	//Sorties
	"DB_BIBLIOTHEQUE".Mobile[#index].Pos[1].Sort1[0] := "I_CP_BD2EVS10_T63";
	"DB_BIBLIOTHEQUE".Mobile[#index].Pos[1].Sort0[0] := "I_CP_BD2EVS10_TVS20";
	"DB_BIBLIOTHEQUE".Mobile[#index].Pos[1].Sort0_Pr_Fin_Pos[0] := "I_CP_BD2EVS10_T63";
	"DB_BIBLIOTHEQUE".Mobile[#index].Pos[1].Sort0_Pr_Fin_Pos[1] := "I_CP_BD2EVS10_TVS20";


	#index := #index + 1;
	(*
	           ╔═══════════╗
	           ║    TR11   ║
	           ╚═══════════╝
	*)
	//++++++++++++++++++++++87++++++++++++++++++++++++++++++\\
	"DB_BIBLIOTHEQUE".Mobile[#index].Noeud := TRUE;

	"DB_BIBLIOTHEQUE".Mobile[#index].Nom := 'TR11';
	"DB_BIBLIOTHEQUE".Mobile[#index].Mob_Suiv[0] := "Index_Mobile"('TR1TR11');
	"DB_BIBLIOTHEQUE".Mobile[#index].Mob_Suiv[1] := "Index_Mobile"('TR2TR11');
	"DB_BIBLIOTHEQUE".Mobile[#index].Mob_Prec[0] := "Index_Mobile"('BD1ER10');
	"DB_BIBLIOTHEQUE".Mobile[#index].Mob_Prec[1] := "Index_Mobile"('BD1EVS10');

	"DB_BIBLIOTHEQUE".Mobile[#index].Pos[0].Nom := '_VERS_TR1TR2TR11';
	"DB_BIBLIOTHEQUE".Mobile[#index].Pos[0].Mob_Suiv[0] := "Index_Mobile"('TR1TR11');
	"DB_BIBLIOTHEQUE".Mobile[#index].Pos[0].Mob_Suiv[1] := "Index_Mobile"('TR2TR11');


	//"DB_BIBLIOTHEQUE".Mobile[#index].Pass_Mat := "RPM_TR11";


	// Entrées avant pos
	"DB_BIBLIOTHEQUE".Mobile[#index].Pos[0].Entr0_Av_Pos[0] := "I_RD_DISJ_TR11";

	// Entrées apres pos
	"DB_BIBLIOTHEQUE".Mobile[#index].Pos[0].Entr0_Ap_Pos[0] := "I_RB_TR11";
	"DB_BIBLIOTHEQUE".Mobile[#index].Pos[0].Entr0_Ap_Pos[1] := "I_RD_DISJ_TR11";


	//"DB_BIBLIOTHEQUE".Mobile[#index].Pos[0].Entr1_Ap_Pos[0] := "I_RR_TR11";
	"DB_BIBLIOTHEQUE".Mobile[#index].Pos[0].Entr1_Ap_Pos[0] := "I_RM_TR11";

	// Entrées fin pos
	//"DB_BIBLIOTHEQUE".Mobile[#index].Pos[0].Entr0_Ap_Fin_Pos[0]:="I_RM_TR11";

	// Sorties
	"DB_BIBLIOTHEQUE".Mobile[#index].Pos[0].Sort1[0] := "I_CM_TR11";
	"DB_BIBLIOTHEQUE".Mobile[#index].Pos[0].Sort0_Pr_Fin_Pos[0] := "I_CM_TR11";


	#index := #index + 1;
	(*
	           ╔═══════════╗
	           ║   TR1TR11 ║
	           ╚═══════════╝
	*)
	//++++++++++++++++++++++88++++++++++++++++++++++++++++++\\



	"DB_BIBLIOTHEQUE".Mobile[#index].Nom := 'TR1TR11';
	"DB_BIBLIOTHEQUE".Mobile[#index].Mob_Suiv[0] := "Index_Mobile"('BD1TR11');
	"DB_BIBLIOTHEQUE".Mobile[#index].Mob_Prec[0] := "Index_Mobile"('TR11');

	"DB_BIBLIOTHEQUE".Mobile[#index].Pos[0].Nom := '_CLOSE';
	//"DB_BIBLIOTHEQUE".Mobile[#index].Pos[0].Mob_Suiv[0] := "Index_Mobile"('BD1TR11');
	"DB_BIBLIOTHEQUE".Mobile[#index].Pos[1].Nom := '_OPEN';
	"DB_BIBLIOTHEQUE".Mobile[#index].Pos[1].Mob_Suiv[0] := "Index_Mobile"('BD1TR11');


	//position fermeture
	"DB_BIBLIOTHEQUE".Mobile[#index].Pos[0].Entr0_Ap_Pos[0] := "I_RPO_TR1TR11";
	"DB_BIBLIOTHEQUE".Mobile[#index].Pos[0].Entr1_Ap_Pos[0] := "I_RPF_TR1TR11";
	"DB_BIBLIOTHEQUE".Mobile[#index].Pos[0].Sort0[0] := "I_CO_TR1TR11";
	"DB_BIBLIOTHEQUE".Mobile[#index].Pos[0].Sort0_Pr_Fin_Pos[0] := "I_CO_TR1TR11";

	//position ouverture
	"DB_BIBLIOTHEQUE".Mobile[#index].Pos[1].Entr0_Ap_Pos[0] := "I_RPF_TR1TR11";
	"DB_BIBLIOTHEQUE".Mobile[#index].Pos[1].Entr1_Ap_Pos[0] := "I_RPO_TR1TR11";
	"DB_BIBLIOTHEQUE".Mobile[#index].Pos[1].Sort1[0] := "I_CO_TR1TR11";
	"DB_BIBLIOTHEQUE".Mobile[#index].Pos[1].Sort0_Pr_Fin_Pos[0] := "I_CO_TR1TR11";



	#index := #index + 1;
	(*
	           ╔═══════════╗
	           ║   TR2TR11 ║
	           ╚═══════════╝
	*)
	//++++++++++++++++++++++89++++++++++++++++++++++++++++++\\


	"DB_BIBLIOTHEQUE".Mobile[#index].Nom := 'TR2TR11';
	"DB_BIBLIOTHEQUE".Mobile[#index].Mob_Suiv[0] := "Index_Mobile"('BD2TR11');
	"DB_BIBLIOTHEQUE".Mobile[#index].Mob_Prec[0] := "Index_Mobile"('TR11');

	"DB_BIBLIOTHEQUE".Mobile[#index].Pos[0].Nom := '_CLOSE';
	//"DB_BIBLIOTHEQUE".Mobile[#index].Pos[0].Mob_Suiv[0] := "Index_Mobile"('BD2TR11');
	"DB_BIBLIOTHEQUE".Mobile[#index].Pos[1].Nom := '_OPEN';
	"DB_BIBLIOTHEQUE".Mobile[#index].Pos[1].Mob_Suiv[0] := "Index_Mobile"('BD2TR11');


	//position fermeture
	"DB_BIBLIOTHEQUE".Mobile[#index].Pos[0].Entr0_Ap_Pos[0] := "I_RPO_TR2TR11";
	"DB_BIBLIOTHEQUE".Mobile[#index].Pos[0].Entr1_Ap_Pos[0] := "I_RPF_TR2TR11";
	"DB_BIBLIOTHEQUE".Mobile[#index].Pos[0].Sort0[0] := "I_CO_TR2TR11";
	"DB_BIBLIOTHEQUE".Mobile[#index].Pos[0].Sort0_Pr_Fin_Pos[0] := "I_CO_TR2TR11";

	//position ouverture
	"DB_BIBLIOTHEQUE".Mobile[#index].Pos[1].Entr0_Ap_Pos[0] := "I_RPF_TR2TR11";
	"DB_BIBLIOTHEQUE".Mobile[#index].Pos[1].Entr1_Ap_Pos[0] := "I_RPO_TR2TR11";
	"DB_BIBLIOTHEQUE".Mobile[#index].Pos[1].Sort1[0] := "I_CO_TR2TR11";
	"DB_BIBLIOTHEQUE".Mobile[#index].Pos[1].Sort0_Pr_Fin_Pos[0] := "I_CO_TR2TR11";



	#index := #index + 1;
	(*
	           ╔═══════════╗
	           ║  BD1TR11  ║
	           ╚═══════════╝
	*)
	//++++++++++++++++++++++90++++++++++++++++++++++++++++++\\
	"DB_BIBLIOTHEQUE".Mobile[#index].Noeud := TRUE;


	"DB_BIBLIOTHEQUE".Mobile[#index].Nom := 'BD1TR11';
	"DB_BIBLIOTHEQUE".Mobile[#index].Mob_Suiv[0] := "Index_Mobile"('S21');
	"DB_BIBLIOTHEQUE".Mobile[#index].Mob_Suiv[1] := "Index_Mobile"('TR12');
	"DB_BIBLIOTHEQUE".Mobile[#index].Mob_Prec[0] := "Index_Mobile"('TR1TR11');


	"DB_BIBLIOTHEQUE".Mobile[#index].Pos[0].Nom := '_VERS_S21';
	"DB_BIBLIOTHEQUE".Mobile[#index].Pos[0].Mob_Suiv[0] := "Index_Mobile"('S21');
	"DB_BIBLIOTHEQUE".Mobile[#index].Pos[1].Nom := '_VERS_TR12';
	"DB_BIBLIOTHEQUE".Mobile[#index].Pos[1].Mob_Suiv[0] := "Index_Mobile"('TR12');




	//Entrées
	"DB_BIBLIOTHEQUE".Mobile[#index].Pos[0].Entr0_Ap_Pos[0] := "I_RP_BD1TR11_TR12";
	"DB_BIBLIOTHEQUE".Mobile[#index].Pos[0].Entr1_Ap_Pos[0] := "I_RP_BD1TR11_S21";
	"DB_BIBLIOTHEQUE".Mobile[#index].Pos[0].Sort1[0] := "I_CP_BD1TR11_S21";
	"DB_BIBLIOTHEQUE".Mobile[#index].Pos[0].Sort0[0] := "I_CP_BD1TR11_TR12";
	"DB_BIBLIOTHEQUE".Mobile[#index].Pos[0].Sort0_Pr_Fin_Pos[0] := "I_CP_BD1TR11_TR12";
	"DB_BIBLIOTHEQUE".Mobile[#index].Pos[0].Sort0_Pr_Fin_Pos[1] := "I_CP_BD1TR11_S21";

	"DB_BIBLIOTHEQUE".Mobile[#index].Pos[1].Entr0_Ap_Pos[1] := "I_RP_BD1TR11_S21";
	"DB_BIBLIOTHEQUE".Mobile[#index].Pos[1].Entr1_Ap_Pos[1] := "I_RP_BD1TR11_TR12";

	//Sorties
	"DB_BIBLIOTHEQUE".Mobile[#index].Pos[1].Sort1[0] := "I_CP_BD1TR11_TR12";
	"DB_BIBLIOTHEQUE".Mobile[#index].Pos[1].Sort0[0] := "I_CP_BD1TR11_S21";
	"DB_BIBLIOTHEQUE".Mobile[#index].Pos[1].Sort0_Pr_Fin_Pos[0] := "I_CP_BD1TR11_TR12";
	"DB_BIBLIOTHEQUE".Mobile[#index].Pos[1].Sort0_Pr_Fin_Pos[1] := "I_CP_BD1TR11_S21";


	#index := #index + 1;
	(*
	           ╔═══════════╗
	           ║  BD2TR11  ║
	           ╚═══════════╝
	*)
	//++++++++++++++++++++++91++++++++++++++++++++++++++++++\\
	"DB_BIBLIOTHEQUE".Mobile[#index].Noeud := TRUE;


	"DB_BIBLIOTHEQUE".Mobile[#index].Nom := 'BD2TR11';
	"DB_BIBLIOTHEQUE".Mobile[#index].Mob_Suiv[0] := "Index_Mobile"('S23');
	"DB_BIBLIOTHEQUE".Mobile[#index].Mob_Suiv[1] := "Index_Mobile"('TR13');
	"DB_BIBLIOTHEQUE".Mobile[#index].Mob_Prec[0] := "Index_Mobile"('TR2TR11');


	"DB_BIBLIOTHEQUE".Mobile[#index].Pos[0].Nom := '_VERS_S23';
	"DB_BIBLIOTHEQUE".Mobile[#index].Pos[0].Mob_Suiv[0] := "Index_Mobile"('S23');
	"DB_BIBLIOTHEQUE".Mobile[#index].Pos[1].Nom := '_VERS_TR13';
	"DB_BIBLIOTHEQUE".Mobile[#index].Pos[1].Mob_Suiv[0] := "Index_Mobile"('TR13');




	//Entrées
	"DB_BIBLIOTHEQUE".Mobile[#index].Pos[0].Entr0_Ap_Pos[0] := "I_RP_BD2TR11_TR13";
	"DB_BIBLIOTHEQUE".Mobile[#index].Pos[0].Entr1_Ap_Pos[0] := "I_RP_BD2TR11_S23";
	"DB_BIBLIOTHEQUE".Mobile[#index].Pos[0].Sort1[0] := "I_CP_BD2TR11_S23";
	"DB_BIBLIOTHEQUE".Mobile[#index].Pos[0].Sort0[0] := "I_CP_BD2TR11_TR13";
	"DB_BIBLIOTHEQUE".Mobile[#index].Pos[0].Sort0_Pr_Fin_Pos[0] := "I_CP_BD2TR11_TR13";
	"DB_BIBLIOTHEQUE".Mobile[#index].Pos[0].Sort0_Pr_Fin_Pos[1] := "I_CP_BD2TR11_S23";

	"DB_BIBLIOTHEQUE".Mobile[#index].Pos[1].Entr0_Ap_Pos[1] := "I_RP_BD2TR11_S23";
	"DB_BIBLIOTHEQUE".Mobile[#index].Pos[1].Entr1_Ap_Pos[1] := "I_RP_BD2TR11_TR13";

	//Sorties
	"DB_BIBLIOTHEQUE".Mobile[#index].Pos[1].Sort1[0] := "I_CP_BD2TR11_TR13";
	"DB_BIBLIOTHEQUE".Mobile[#index].Pos[1].Sort0[0] := "I_CP_BD2TR11_S23";
	"DB_BIBLIOTHEQUE".Mobile[#index].Pos[1].Sort0_Pr_Fin_Pos[0] := "I_CP_BD2TR11_TR13";
	"DB_BIBLIOTHEQUE".Mobile[#index].Pos[1].Sort0_Pr_Fin_Pos[1] := "I_CP_BD2TR11_S23";


	#index := #index + 1;
	(*
	           ╔═══════════╗
	           ║    TR12   ║
	           ╚═══════════╝
	*)
	//++++++++++++++++++++++92++++++++++++++++++++++++++++++\\


	"DB_BIBLIOTHEQUE".Mobile[#index].Nom := 'TR12';
	"DB_BIBLIOTHEQUE".Mobile[#index].Mob_Suiv[0] := "Index_Mobile"('S22');
	"DB_BIBLIOTHEQUE".Mobile[#index].Mob_Prec[0] := "Index_Mobile"('BD1TR11');

	"DB_BIBLIOTHEQUE".Mobile[#index].Pos[0].Nom := '_VERSS22';
	"DB_BIBLIOTHEQUE".Mobile[#index].Pos[0].Mob_Suiv[0] := "Index_Mobile"('S22');


	//"DB_BIBLIOTHEQUE".Mobile[#index].Pass_Mat := "RPM_TR12";


	// Entrées avant pos
	"DB_BIBLIOTHEQUE".Mobile[#index].Pos[0].Entr0_Av_Pos[0] := "I_RD_DISJ_TR12";

	// Entrées apres pos
	"DB_BIBLIOTHEQUE".Mobile[#index].Pos[0].Entr0_Ap_Pos[0] := "I_RB_TR12";
	"DB_BIBLIOTHEQUE".Mobile[#index].Pos[0].Entr0_Ap_Pos[1] := "I_RD_DISJ_TR12";


	//"DB_BIBLIOTHEQUE".Mobile[#index].Pos[0].Entr1_Ap_Pos[0] := "I_RR_TR12";
	"DB_BIBLIOTHEQUE".Mobile[#index].Pos[0].Entr1_Ap_Pos[0] := "I_RM_TR12";

	// Entrées fin pos
	//"DB_BIBLIOTHEQUE".Mobile[#index].Pos[0].Entr0_Ap_Fin_Pos[0]:="I_RM_TR12";

	// Sorties
	"DB_BIBLIOTHEQUE".Mobile[#index].Pos[0].Sort1[0] := "I_CM_TR12";
	"DB_BIBLIOTHEQUE".Mobile[#index].Pos[0].Sort0_Pr_Fin_Pos[0] := "I_CM_TR12";


	#index := #index + 1;
	(*
	           ╔═══════════╗
	           ║    TR13   ║
	           ╚═══════════╝
	*)
	//++++++++++++++++++++++93++++++++++++++++++++++++++++++\\


	"DB_BIBLIOTHEQUE".Mobile[#index].Nom := 'TR13';
	"DB_BIBLIOTHEQUE".Mobile[#index].Mob_Suiv[0] := "Index_Mobile"('S24');
	"DB_BIBLIOTHEQUE".Mobile[#index].Mob_Prec[0] := "Index_Mobile"('BD2TR11');

	"DB_BIBLIOTHEQUE".Mobile[#index].Pos[0].Nom := '_VERSS24';
	"DB_BIBLIOTHEQUE".Mobile[#index].Pos[0].Mob_Suiv[0] := "Index_Mobile"('S24');

	//"DB_BIBLIOTHEQUE".Mobile[#index].Pass_Mat := "RPM_TR13";


	// Entrées avant pos
	"DB_BIBLIOTHEQUE".Mobile[#index].Pos[0].Entr0_Av_Pos[0] := "I_RD_DISJ_TR13";

	// Entrées apres pos
	"DB_BIBLIOTHEQUE".Mobile[#index].Pos[0].Entr0_Ap_Pos[0] := "I_RB_TR13";
	"DB_BIBLIOTHEQUE".Mobile[#index].Pos[0].Entr0_Ap_Pos[1] := "I_RD_DISJ_TR13";


	//"DB_BIBLIOTHEQUE".Mobile[#index].Pos[0].Entr1_Ap_Pos[0] := "I_RR_TR13";
	"DB_BIBLIOTHEQUE".Mobile[#index].Pos[0].Entr1_Ap_Pos[0] := "I_RM_TR13";

	// Entrées fin pos
	//"DB_BIBLIOTHEQUE".Mobile[#index].Pos[0].Entr0_Ap_Fin_Pos[0]:="I_RM_TR13";

	// Sorties
	"DB_BIBLIOTHEQUE".Mobile[#index].Pos[0].Sort1[0] := "I_CM_TR13";
	"DB_BIBLIOTHEQUE".Mobile[#index].Pos[0].Sort0_Pr_Fin_Pos[0] := "I_CM_TR13";


	#index := #index + 1;
	(*
	           ╔═══════════╗
	           ║   VAS21   ║
	           ╚═══════════╝
	*)
	//++++++++++++++++++++++94++++++++++++++++++++++++++++++\\



	"DB_BIBLIOTHEQUE".Mobile[#index].Nom := 'VAS21';
	"DB_BIBLIOTHEQUE".Mobile[#index].Mob_Suiv[0] := "Index_Mobile"('TVS212');
	"DB_BIBLIOTHEQUE".Mobile[#index].Mob_Prec[0] := "Index_Mobile"('S21');

	"DB_BIBLIOTHEQUE".Mobile[#index].Pos[0].Nom := '_CLOSE';
	//"DB_BIBLIOTHEQUE".Mobile[#index].Pos[0].Mob_Suiv[0] := "Index_Mobile"('TVS212');
	"DB_BIBLIOTHEQUE".Mobile[#index].Pos[1].Nom := '_OPEN';
	"DB_BIBLIOTHEQUE".Mobile[#index].Pos[1].Mob_Suiv[0] := "Index_Mobile"('TVS212');


	//position fermeture
	"DB_BIBLIOTHEQUE".Mobile[#index].Pos[0].Entr0_Ap_Pos[0] := "I_RPO_VAS21";
	"DB_BIBLIOTHEQUE".Mobile[#index].Pos[0].Entr1_Ap_Pos[0] := "I_RPF_VAS21";
	"DB_BIBLIOTHEQUE".Mobile[#index].Pos[0].Sort0[0] := "I_CO_VAS21";
	"DB_BIBLIOTHEQUE".Mobile[#index].Pos[0].Sort0_Pr_Fin_Pos[0] := "I_CO_VAS21";

	//position ouverture
	"DB_BIBLIOTHEQUE".Mobile[#index].Pos[1].Entr0_Ap_Pos[0] := "I_RPF_VAS21";
	"DB_BIBLIOTHEQUE".Mobile[#index].Pos[1].Entr1_Ap_Pos[0] := "I_RPO_VAS21";
	"DB_BIBLIOTHEQUE".Mobile[#index].Pos[1].Sort1[0] := "I_CO_VAS21";
	"DB_BIBLIOTHEQUE".Mobile[#index].Pos[1].Sort0_Pr_Fin_Pos[0] := "I_CO_VAS21";



	#index := #index + 1;

	(*
	           ╔═══════════╗
	           ║   VAS22   ║
	           ╚═══════════╝
	*)
	//++++++++++++++++++++++95++++++++++++++++++++++++++++++\\



	"DB_BIBLIOTHEQUE".Mobile[#index].Nom := 'VAS22';
	"DB_BIBLIOTHEQUE".Mobile[#index].Mob_Suiv[0] := "Index_Mobile"('TVS22');
	"DB_BIBLIOTHEQUE".Mobile[#index].Mob_Prec[0] := "Index_Mobile"('S22');

	"DB_BIBLIOTHEQUE".Mobile[#index].Pos[0].Nom := '_CLOSE';
	//"DB_BIBLIOTHEQUE".Mobile[#index].Pos[0].Mob_Suiv[0] := "Index_Mobile"('TVS22');
	"DB_BIBLIOTHEQUE".Mobile[#index].Pos[1].Nom := '_OPEN';
	"DB_BIBLIOTHEQUE".Mobile[#index].Pos[1].Mob_Suiv[0] := "Index_Mobile"('TVS22');


	//position fermeture
	"DB_BIBLIOTHEQUE".Mobile[#index].Pos[0].Entr0_Ap_Pos[0] := "I_RPO_VAS22";
	"DB_BIBLIOTHEQUE".Mobile[#index].Pos[0].Entr1_Ap_Pos[0] := "I_RPF_VAS22";
	"DB_BIBLIOTHEQUE".Mobile[#index].Pos[0].Sort0[0] := "I_CO_VAS22";
	"DB_BIBLIOTHEQUE".Mobile[#index].Pos[0].Sort0_Pr_Fin_Pos[0] := "I_CO_VAS22";

	//position ouverture
	"DB_BIBLIOTHEQUE".Mobile[#index].Pos[1].Entr0_Ap_Pos[0] := "I_RPF_VAS22";
	"DB_BIBLIOTHEQUE".Mobile[#index].Pos[1].Entr1_Ap_Pos[0] := "I_RPO_VAS22";
	"DB_BIBLIOTHEQUE".Mobile[#index].Pos[1].Sort1[0] := "I_CO_VAS22";
	"DB_BIBLIOTHEQUE".Mobile[#index].Pos[1].Sort0_Pr_Fin_Pos[0] := "I_CO_VAS22";



	#index := #index + 1;
	(*
	           ╔═══════════╗
	           ║   VAS23   ║
	           ╚═══════════╝
	*)
	//++++++++++++++++++++++96++++++++++++++++++++++++++++++\\



	"DB_BIBLIOTHEQUE".Mobile[#index].Nom := 'VAS23';
	"DB_BIBLIOTHEQUE".Mobile[#index].Mob_Suiv[0] := "Index_Mobile"('TVS212');
	"DB_BIBLIOTHEQUE".Mobile[#index].Mob_Prec[0] := "Index_Mobile"('S23');

	"DB_BIBLIOTHEQUE".Mobile[#index].Pos[0].Nom := '_CLOSE';
	//"DB_BIBLIOTHEQUE".Mobile[#index].Pos[0].Mob_Suiv[0] := "Index_Mobile"('TVS212');
	"DB_BIBLIOTHEQUE".Mobile[#index].Pos[1].Nom := '_OPEN';
	"DB_BIBLIOTHEQUE".Mobile[#index].Pos[1].Mob_Suiv[0] := "Index_Mobile"('TVS212');


	//position fermeture
	"DB_BIBLIOTHEQUE".Mobile[#index].Pos[0].Entr0_Ap_Pos[0] := "I_RPO_VAS23";
	"DB_BIBLIOTHEQUE".Mobile[#index].Pos[0].Entr1_Ap_Pos[0] := "I_RPF_VAS23";
	"DB_BIBLIOTHEQUE".Mobile[#index].Pos[0].Sort0[0] := "I_CO_VAS23";
	"DB_BIBLIOTHEQUE".Mobile[#index].Pos[0].Sort0_Pr_Fin_Pos[0] := "I_CO_VAS23";

	//position ouverture
	"DB_BIBLIOTHEQUE".Mobile[#index].Pos[1].Entr0_Ap_Pos[0] := "I_RPF_VAS23";
	"DB_BIBLIOTHEQUE".Mobile[#index].Pos[1].Entr1_Ap_Pos[0] := "I_RPO_VAS23";
	"DB_BIBLIOTHEQUE".Mobile[#index].Pos[1].Sort1[0] := "I_CO_VAS23";
	"DB_BIBLIOTHEQUE".Mobile[#index].Pos[1].Sort0_Pr_Fin_Pos[0] := "I_CO_VAS23";



	#index := #index + 1;
	(*
	           ╔═══════════╗
	           ║   VAS24   ║
	           ╚═══════════╝
	*)
	//++++++++++++++++++++++97++++++++++++++++++++++++++++++\\



	"DB_BIBLIOTHEQUE".Mobile[#index].Nom := 'VAS24';
	"DB_BIBLIOTHEQUE".Mobile[#index].Mob_Suiv[0] := "Index_Mobile"('TVS24');
	"DB_BIBLIOTHEQUE".Mobile[#index].Mob_Prec[0] := "Index_Mobile"('S24');

	"DB_BIBLIOTHEQUE".Mobile[#index].Pos[0].Nom := '_CLOSE';
	//"DB_BIBLIOTHEQUE".Mobile[#index].Pos[0].Mob_Suiv[0] := "Index_Mobile"('TVS24');
	"DB_BIBLIOTHEQUE".Mobile[#index].Pos[1].Nom := '_OPEN';
	"DB_BIBLIOTHEQUE".Mobile[#index].Pos[1].Mob_Suiv[0] := "Index_Mobile"('TVS24');


	//position fermeture
	"DB_BIBLIOTHEQUE".Mobile[#index].Pos[0].Entr0_Ap_Pos[0] := "I_RPO_VAS24";
	"DB_BIBLIOTHEQUE".Mobile[#index].Pos[0].Entr1_Ap_Pos[0] := "I_RPF_VAS24";
	"DB_BIBLIOTHEQUE".Mobile[#index].Pos[0].Sort0[0] := "I_CO_VAS24";
	"DB_BIBLIOTHEQUE".Mobile[#index].Pos[0].Sort0_Pr_Fin_Pos[0] := "I_CO_VAS24";

	//position ouverture
	"DB_BIBLIOTHEQUE".Mobile[#index].Pos[1].Entr0_Ap_Pos[0] := "I_RPF_VAS24";
	"DB_BIBLIOTHEQUE".Mobile[#index].Pos[1].Entr1_Ap_Pos[0] := "I_RPO_VAS24";
	"DB_BIBLIOTHEQUE".Mobile[#index].Pos[1].Sort1[0] := "I_CO_VAS24";
	"DB_BIBLIOTHEQUE".Mobile[#index].Pos[1].Sort0_Pr_Fin_Pos[0] := "I_CO_VAS24";



	#index := #index + 1;
	(*
	           ╔═══════════╗
	           ║   TVS22   ║
	           ╚═══════════╝
	*)
	//++++++++++++++++++++++98++++++++++++++++++++++++++++++\\


	"DB_BIBLIOTHEQUE".Mobile[#index].Nom := 'TVS22';
	"DB_BIBLIOTHEQUE".Mobile[#index].Mob_Suiv[0] := "Index_Mobile"('TVS212');
	"DB_BIBLIOTHEQUE".Mobile[#index].Mob_Prec[0] := "Index_Mobile"('S22');

	"DB_BIBLIOTHEQUE".Mobile[#index].Pos[0].Nom := '_VERSTVS212';
	"DB_BIBLIOTHEQUE".Mobile[#index].Pos[0].Mob_Suiv[0] := "Index_Mobile"('TVS212');

	//"DB_BIBLIOTHEQUE".Mobile[#index].Pass_Mat := "RPM_TVS22";


	// Entrées avant pos
	"DB_BIBLIOTHEQUE".Mobile[#index].Pos[0].Entr0_Av_Pos[0] := "I_RD_DISJ_TVS22";

	// Entrées apres pos
	//"DB_BIBLIOTHEQUE".Mobile[#index].Pos[0].Entr0_Ap_Pos[0] := "I_RB_TVS22";
	"DB_BIBLIOTHEQUE".Mobile[#index].Pos[0].Entr0_Ap_Pos[0] := "I_RD_DISJ_TVS22";


	//"DB_BIBLIOTHEQUE".Mobile[#index].Pos[0].Entr1_Ap_Pos[0] := "I_RR_TVS22";
	"DB_BIBLIOTHEQUE".Mobile[#index].Pos[0].Entr1_Ap_Pos[0] := "I_RM_TVS22";

	// Entrées fin pos
	//"DB_BIBLIOTHEQUE".Mobile[#index].Pos[0].Entr0_Ap_Fin_Pos[0]:="I_RM_TVS22";

	// Sorties
	"DB_BIBLIOTHEQUE".Mobile[#index].Pos[0].Sort1[0] := "I_CM_TVS22";
	"DB_BIBLIOTHEQUE".Mobile[#index].Pos[0].Sort0_Pr_Fin_Pos[0] := "I_CM_TVS22";


	#index := #index + 1;
	(*
	           ╔═══════════╗
	           ║   TVS24   ║
	           ╚═══════════╝
	*)
	//++++++++++++++++++++++99++++++++++++++++++++++++++++++\\


	"DB_BIBLIOTHEQUE".Mobile[#index].Nom := 'TVS24';
	"DB_BIBLIOTHEQUE".Mobile[#index].Mob_Suiv[0] := "Index_Mobile"('TVS212');
	"DB_BIBLIOTHEQUE".Mobile[#index].Mob_Prec[0] := "Index_Mobile"('S24');

	"DB_BIBLIOTHEQUE".Mobile[#index].Pos[0].Nom := '_VERSTVS212';
	"DB_BIBLIOTHEQUE".Mobile[#index].Pos[0].Mob_Suiv[0] := "Index_Mobile"('TVS212');

	//"DB_BIBLIOTHEQUE".Mobile[#index].Pass_Mat := "RPM_TVS24";


	// Entrées avant pos
	"DB_BIBLIOTHEQUE".Mobile[#index].Pos[0].Entr0_Av_Pos[0] := "I_RD_DISJ_TVS24";

	// Entrées apres pos
	"DB_BIBLIOTHEQUE".Mobile[#index].Pos[0].Entr0_Ap_Pos[0] := "I_RB_TVS24";
	"DB_BIBLIOTHEQUE".Mobile[#index].Pos[0].Entr0_Ap_Pos[1] := "I_RD_DISJ_TVS24";


	//"DB_BIBLIOTHEQUE".Mobile[#index].Pos[0].Entr1_Ap_Pos[0] := "I_RR_TVS24";
	"DB_BIBLIOTHEQUE".Mobile[#index].Pos[0].Entr1_Ap_Pos[0] := "I_RM_TVS24";

	// Entrées fin pos
	//"DB_BIBLIOTHEQUE".Mobile[#index].Pos[0].Entr0_Ap_Fin_Pos[0]:="I_RM_TVS24";

	// Sorties
	"DB_BIBLIOTHEQUE".Mobile[#index].Pos[0].Sort1[0] := "I_CM_TVS24";
	"DB_BIBLIOTHEQUE".Mobile[#index].Pos[0].Sort0_Pr_Fin_Pos[0] := "I_CM_TVS24";


	#index := #index + 1;
	(*
	           ╔═══════════╗
	           ║   TVS212  ║
	           ╚═══════════╝
	*)
	//++++++++++++++++++++++100++++++++++++++++++++++++++++++\\


	"DB_BIBLIOTHEQUE".Mobile[#index].Nom := 'TVS212';
	"DB_BIBLIOTHEQUE".Mobile[#index].Mob_Suiv[0] := "Index_Mobile"('BDTVS');
	"DB_BIBLIOTHEQUE".Mobile[#index].Mob_Prec[0] := "Index_Mobile"('TVS24');
	"DB_BIBLIOTHEQUE".Mobile[#index].Mob_Prec[1] := "Index_Mobile"('VAS23');
	"DB_BIBLIOTHEQUE".Mobile[#index].Mob_Prec[2] := "Index_Mobile"('TVS22');
	"DB_BIBLIOTHEQUE".Mobile[#index].Mob_Prec[3] := "Index_Mobile"('VAS21');

	"DB_BIBLIOTHEQUE".Mobile[#index].Pos[0].Nom := '_VERS_BDTVS';
	"DB_BIBLIOTHEQUE".Mobile[#index].Pos[0].Mob_Suiv[0] := "Index_Mobile"('BDTVS');

	//"DB_BIBLIOTHEQUE".Mobile[#index].Pass_Mat := "RPM_TVS212";


	// Entrées avant pos
	"DB_BIBLIOTHEQUE".Mobile[#index].Pos[0].Entr0_Av_Pos[0] := "I_RD_DISJ_TVS212";

	// Entrées apres pos
	"DB_BIBLIOTHEQUE".Mobile[#index].Pos[0].Entr0_Ap_Pos[0] := "I_RB_TVS212";
	"DB_BIBLIOTHEQUE".Mobile[#index].Pos[0].Entr0_Ap_Pos[1] := "I_RD_DISJ_TVS212";


	//"DB_BIBLIOTHEQUE".Mobile[#index].Pos[0].Entr1_Ap_Pos[0] := "I_RR_TVS212";
	"DB_BIBLIOTHEQUE".Mobile[#index].Pos[0].Entr1_Ap_Pos[0] := "I_RM_TVS212";

	// Entrées fin pos
	//"DB_BIBLIOTHEQUE".Mobile[#index].Pos[0].Entr0_Ap_Fin_Pos[0]:="I_RM_TVS212";

	// Sorties
	"DB_BIBLIOTHEQUE".Mobile[#index].Pos[0].Sort1[0] := "I_CM_TVS212";
	"DB_BIBLIOTHEQUE".Mobile[#index].Pos[0].Sort0_Pr_Fin_Pos[0] := "I_CM_TVS212";

	#index := #index + 1;
	(*
	           ╔═══════════╗
	           ║   TVS20   ║
	           ╚═══════════╝
	*)
	//++++++++++++++++++++++101++++++++++++++++++++++++++++++\\
	"DB_BIBLIOTHEQUE".Mobile[#index].Noeud := TRUE;

	"DB_BIBLIOTHEQUE".Mobile[#index].Nom := 'TVS20';
	"DB_BIBLIOTHEQUE".Mobile[#index].Mob_Suiv[0] := "Index_Mobile"('TR1TVS20');
	"DB_BIBLIOTHEQUE".Mobile[#index].Mob_Suiv[1] := "Index_Mobile"('TR2TVS20');
	"DB_BIBLIOTHEQUE".Mobile[#index].Mob_Prec[0] := "Index_Mobile"('BD2EVS10');

	"DB_BIBLIOTHEQUE".Mobile[#index].Pos[0].Nom := '_VERS_B1_B2';
	"DB_BIBLIOTHEQUE".Mobile[#index].Pos[0].Mob_Suiv[0] := "Index_Mobile"('TR1TVS20');
	"DB_BIBLIOTHEQUE".Mobile[#index].Pos[0].Mob_Suiv[1] := "Index_Mobile"('TR2TVS20');

	//"DB_BIBLIOTHEQUE".Mobile[#index].Pass_Mat := "RPM_TVS20";


	// Entrées avant pos
	"DB_BIBLIOTHEQUE".Mobile[#index].Pos[0].Entr0_Av_Pos[0] := "I_RD_DISJ_TVS20";

	// Entrées apres pos
	"DB_BIBLIOTHEQUE".Mobile[#index].Pos[0].Entr0_Ap_Pos[0] := "I_RB_TVS20";
	"DB_BIBLIOTHEQUE".Mobile[#index].Pos[0].Entr0_Ap_Pos[1] := "I_RD_DISJ_TVS20";


	//"DB_BIBLIOTHEQUE".Mobile[#index].Pos[0].Entr1_Ap_Pos[0] := "I_RR_TVS20";
	"DB_BIBLIOTHEQUE".Mobile[#index].Pos[0].Entr1_Ap_Pos[0] := "I_RM_TVS20";

	// Entrées fin pos
	//"DB_BIBLIOTHEQUE".Mobile[#index].Pos[0].Entr0_Ap_Fin_Pos[0]:="I_RM_TVS20";

	// Sorties
	"DB_BIBLIOTHEQUE".Mobile[#index].Pos[0].Sort1[0] := "I_CM_TVS20";
	"DB_BIBLIOTHEQUE".Mobile[#index].Pos[0].Sort0_Pr_Fin_Pos[0] := "I_CM_TVS20";


	#index := #index + 1;
	(*
	           ╔═══════════╗
	           ║  TR1TVS20 ║
	           ╚═══════════╝
	*)
	//++++++++++++++++++++++102++++++++++++++++++++++++++++++\\



	"DB_BIBLIOTHEQUE".Mobile[#index].Nom := 'TR1TVS20';
	"DB_BIBLIOTHEQUE".Mobile[#index].Mob_Suiv[0] := "Index_Mobile"('B01');
	"DB_BIBLIOTHEQUE".Mobile[#index].Mob_Prec[0] := "Index_Mobile"('TVS20');

	"DB_BIBLIOTHEQUE".Mobile[#index].Pos[0].Nom := '_CLOSE';
	//"DB_BIBLIOTHEQUE".Mobile[#index].Pos[0].Mob_Suiv[0] := "Index_Mobile"('B01');
	"DB_BIBLIOTHEQUE".Mobile[#index].Pos[1].Nom := '_OPEN';
	"DB_BIBLIOTHEQUE".Mobile[#index].Pos[1].Mob_Suiv[0] := "Index_Mobile"('B01');


	//position fermeture
	"DB_BIBLIOTHEQUE".Mobile[#index].Pos[0].Entr0_Ap_Pos[0] := "I_RPO_TR1TVS20";
	"DB_BIBLIOTHEQUE".Mobile[#index].Pos[0].Entr1_Ap_Pos[0] := "I_RPF_TR1TVS20";
	"DB_BIBLIOTHEQUE".Mobile[#index].Pos[0].Sort0[0] := "I_CO_TR1TVS20";
	"DB_BIBLIOTHEQUE".Mobile[#index].Pos[0].Sort0_Pr_Fin_Pos[0] := "I_CO_TR1TVS20";

	//position ouverture
	"DB_BIBLIOTHEQUE".Mobile[#index].Pos[1].Entr0_Ap_Pos[0] := "I_RPF_TR1TVS20";
	"DB_BIBLIOTHEQUE".Mobile[#index].Pos[1].Entr1_Ap_Pos[0] := "I_RPO_TR1TVS20";
	"DB_BIBLIOTHEQUE".Mobile[#index].Pos[1].Sort1[0] := "I_CO_TR1TVS20";
	"DB_BIBLIOTHEQUE".Mobile[#index].Pos[1].Sort0_Pr_Fin_Pos[0] := "I_CO_TR1TVS20";



	#index := #index + 1;
	(*
	           ╔═══════════╗
	           ║  TR2TVS20 ║
	           ╚═══════════╝
	*)
	//++++++++++++++++++++++103++++++++++++++++++++++++++++++\\



	"DB_BIBLIOTHEQUE".Mobile[#index].Nom := 'TR2TVS20';
	"DB_BIBLIOTHEQUE".Mobile[#index].Mob_Suiv[0] := "Index_Mobile"('B02');
	"DB_BIBLIOTHEQUE".Mobile[#index].Mob_Prec[0] := "Index_Mobile"('TVS20');

	"DB_BIBLIOTHEQUE".Mobile[#index].Pos[0].Nom := '_CLOSE';
	//"DB_BIBLIOTHEQUE".Mobile[#index].Pos[0].Mob_Suiv[0] := "Index_Mobile"('B02');
	"DB_BIBLIOTHEQUE".Mobile[#index].Pos[1].Nom := '_OPEN';
	"DB_BIBLIOTHEQUE".Mobile[#index].Pos[1].Mob_Suiv[0] := "Index_Mobile"('B02');


	//position fermeture
	"DB_BIBLIOTHEQUE".Mobile[#index].Pos[0].Entr0_Ap_Pos[0] := "I_RPO_TR2TVS20";
	"DB_BIBLIOTHEQUE".Mobile[#index].Pos[0].Entr1_Ap_Pos[0] := "I_RPF_TR2TVS20";
	"DB_BIBLIOTHEQUE".Mobile[#index].Pos[0].Sort0[0] := "I_CO_TR2TVS20";
	"DB_BIBLIOTHEQUE".Mobile[#index].Pos[0].Sort0_Pr_Fin_Pos[0] := "I_CO_TR2TVS20";

	//position ouverture
	"DB_BIBLIOTHEQUE".Mobile[#index].Pos[1].Entr0_Ap_Pos[0] := "I_RPF_TR2TVS20";
	"DB_BIBLIOTHEQUE".Mobile[#index].Pos[1].Entr1_Ap_Pos[0] := "I_RPO_TR2TVS20";
	"DB_BIBLIOTHEQUE".Mobile[#index].Pos[1].Sort1[0] := "I_CO_TR2TVS20";
	"DB_BIBLIOTHEQUE".Mobile[#index].Pos[1].Sort0_Pr_Fin_Pos[0] := "I_CO_TR2TVS20";



	#index := #index + 1;
	(*
	           ╔═══════════╗
	           ║  TR1T63   ║
	           ╚═══════════╝
	*)
	//++++++++++++++++++++++104++++++++++++++++++++++++++++++\\



	"DB_BIBLIOTHEQUE".Mobile[#index].Nom := 'TR1T63';
	"DB_BIBLIOTHEQUE".Mobile[#index].Mob_Suiv[0] := "Index_Mobile"('T02');
	"DB_BIBLIOTHEQUE".Mobile[#index].Mob_Prec[0] := "Index_Mobile"('T63');

	"DB_BIBLIOTHEQUE".Mobile[#index].Pos[0].Nom := '_CLOSE';
	//"DB_BIBLIOTHEQUE".Mobile[#index].Pos[0].Mob_Suiv[0] := "Index_Mobile"('T02');
	"DB_BIBLIOTHEQUE".Mobile[#index].Pos[1].Nom := '_OPEN';
	"DB_BIBLIOTHEQUE".Mobile[#index].Pos[1].Mob_Suiv[0] := "Index_Mobile"('T02');


	//position fermeture
	"DB_BIBLIOTHEQUE".Mobile[#index].Pos[0].Entr0_Ap_Pos[0] := "I_RPO_TR1T63";
	"DB_BIBLIOTHEQUE".Mobile[#index].Pos[0].Entr1_Ap_Pos[0] := "I_RPF_TR1T63";
	"DB_BIBLIOTHEQUE".Mobile[#index].Pos[0].Sort0[0] := "I_CO_TR1T63";
	"DB_BIBLIOTHEQUE".Mobile[#index].Pos[0].Sort0_Pr_Fin_Pos[0] := "I_CO_TR1T63";

	//position ouverture
	"DB_BIBLIOTHEQUE".Mobile[#index].Pos[1].Entr0_Ap_Pos[0] := "I_RPF_TR1T63";
	"DB_BIBLIOTHEQUE".Mobile[#index].Pos[1].Entr1_Ap_Pos[0] := "I_RPO_TR1T63";
	"DB_BIBLIOTHEQUE".Mobile[#index].Pos[1].Sort1[0] := "I_CO_TR1T63";
	"DB_BIBLIOTHEQUE".Mobile[#index].Pos[1].Sort0_Pr_Fin_Pos[0] := "I_CO_TR1T63";



	#index := #index + 1;
	(*
	           ╔═══════════╗
	           ║  VisS21   ║
	           ╚═══════════╝
	*)
	//++++++++++++++++++++++105++++++++++++++++++++++++++++++\\
	"DB_BIBLIOTHEQUE".Mobile[#index].Nom := 'VisS21';





	"DB_BIBLIOTHEQUE".Mobile[#index].Tjr_Desasservi := TRUE;


	// Entrées avant pos
	"DB_BIBLIOTHEQUE".Mobile[#index].Pos[0].Entr0_Av_Pos[0] := "I_RD_DISJ_VIS21";
	// Entrées apres pos
	"DB_BIBLIOTHEQUE".Mobile[#index].Pos[0].Entr0_Ap_Pos[1] := "I_RD_DISJ_VIS21";
	"DB_BIBLIOTHEQUE".Mobile[#index].Pos[0].Entr1_Ap_Pos[1] := "I_RM_VIS21";

	// Entrées fin pos
	//"DB_BIBLIOTHEQUE".Mobile[#index].Pos[0].Entr0_Ap_Fin_Pos[0]:="I_RM_VisS21";

	// Sorties
	"DB_BIBLIOTHEQUE".Mobile[#index].Pos[0].Sort1[0] := "I_CM_VIS21";
	"DB_BIBLIOTHEQUE".Mobile[#index].Pos[0].Sort0_Pr_Fin_Pos[0] := "I_CM_VIS21";
	#index := #index + 1;



	(*
	           ╔═══════════╗
	           ║  VisS22   ║
	           ╚═══════════╝
	*)
	//++++++++++++++++++++++106++++++++++++++++++++++++++++++\\
	"DB_BIBLIOTHEQUE".Mobile[#index].Nom := 'VisS22';





	"DB_BIBLIOTHEQUE".Mobile[#index].Tjr_Desasservi := TRUE;

	// Entrées avant pos
	"DB_BIBLIOTHEQUE".Mobile[#index].Pos[0].Entr0_Av_Pos[0] := "I_RD_DISJ_VIS22";
	// Entrées apres pos
	"DB_BIBLIOTHEQUE".Mobile[#index].Pos[0].Entr0_Ap_Pos[1] := "I_RD_DISJ_VIS22";
	"DB_BIBLIOTHEQUE".Mobile[#index].Pos[0].Entr1_Ap_Pos[1] := "I_RM_VIS22";

	// Entrées fin pos
	//"DB_BIBLIOTHEQUE".Mobile[#index].Pos[0].Entr0_Ap_Fin_Pos[0]:="I_RM_ViS22";

	// Sorties
	"DB_BIBLIOTHEQUE".Mobile[#index].Pos[0].Sort1[0] := "I_CM_VIS22";
	"DB_BIBLIOTHEQUE".Mobile[#index].Pos[0].Sort0_Pr_Fin_Pos[0] := "I_CM_VIS22";
	#index := #index + 1;
	(*
	           ╔═══════════╗
	           ║  VisS23   ║
	           ╚═══════════╝
	*)
	//++++++++++++++++++++++107++++++++++++++++++++++++++++++\\
	"DB_BIBLIOTHEQUE".Mobile[#index].Nom := 'VisS23';





	"DB_BIBLIOTHEQUE".Mobile[#index].Tjr_Desasservi := TRUE;

	// Entrées avant pos
	"DB_BIBLIOTHEQUE".Mobile[#index].Pos[0].Entr0_Av_Pos[0] := "I_RD_DISJ_VIS23";
	// Entrées apres pos
	"DB_BIBLIOTHEQUE".Mobile[#index].Pos[0].Entr0_Ap_Pos[1] := "I_RD_DISJ_VIS23";
	"DB_BIBLIOTHEQUE".Mobile[#index].Pos[0].Entr1_Ap_Pos[1] := "I_RM_VIS23";

	// Entrées fin pos
	//"DB_BIBLIOTHEQUE".Mobile[#index].Pos[0].Entr0_Ap_Fin_Pos[0]:="I_RM_ViS23";

	// Sorties
	"DB_BIBLIOTHEQUE".Mobile[#index].Pos[0].Sort1[0] := "I_CM_VIS23";
	"DB_BIBLIOTHEQUE".Mobile[#index].Pos[0].Sort0_Pr_Fin_Pos[0] := "I_CM_VIS23";
	#index := #index + 1;
	(*
	           ╔═══════════╗
	           ║  VisS24   ║
	           ╚═══════════╝
	*)
	//++++++++++++++++++++++108++++++++++++++++++++++++++++++\\
	"DB_BIBLIOTHEQUE".Mobile[#index].Nom := 'VisS24';





	"DB_BIBLIOTHEQUE".Mobile[#index].Tjr_Desasservi := TRUE;

	// Entrées avant pos
	"DB_BIBLIOTHEQUE".Mobile[#index].Pos[0].Entr0_Av_Pos[0] := "I_RD_DISJ_VIS24";
	// Entrées apres pos
	"DB_BIBLIOTHEQUE".Mobile[#index].Pos[0].Entr0_Ap_Pos[1] := "I_RD_DISJ_VIS24";
	"DB_BIBLIOTHEQUE".Mobile[#index].Pos[0].Entr1_Ap_Pos[1] := "I_RM_VIS24";

	// Entrées fin pos
	//"DB_BIBLIOTHEQUE".Mobile[#index].Pos[0].Entr0_Ap_Fin_Pos[0]:="I_RM_ViS24";

	// Sorties
	"DB_BIBLIOTHEQUE".Mobile[#index].Pos[0].Sort1[0] := "I_CM_VIS24";
	"DB_BIBLIOTHEQUE".Mobile[#index].Pos[0].Sort0_Pr_Fin_Pos[0] := "I_CM_VIS24";
	#index := #index + 1;
	(*
	           ╔═══════════╗
	           ║    BV01   ║
	           ╚═══════════╝
	*)
	//++++++++++++++++++++++109++++++++++++++++++++++++++++++\\
	"DB_BIBLIOTHEQUE".Mobile[#index].Nom := 'BV01';





	#index := #index + 1;
	(*
	           ╔═══════════╗
	           ║   TRBV01  ║
	           ╚═══════════╝
	*)
	//++++++++++++++++++++++110++++++++++++++++++++++++++++++\\

	"DB_BIBLIOTHEQUE".Mobile[#index].Nom := 'TRBV01';
	"DB_BIBLIOTHEQUE".Mobile[#index].Mob_Prec[0] := "Index_Mobile"('BV01');
	"DB_BIBLIOTHEQUE".Mobile[#index].Tjr_Desasservi := TRUE;
	"DB_BIBLIOTHEQUE".Mobile[#index].Asservi := FALSE;
	"DB_BIBLIOTHEQUE".Mobile[#index].Pos[0].Nom := '_CLOSE';
	"DB_BIBLIOTHEQUE".Mobile[#index].Pos[1].Nom := '_OPEN';

	//position fermeture
	"DB_BIBLIOTHEQUE".Mobile[#index].Pos[0].Entr0_Ap_Pos[0] := "I_RPO_TRBV01";
	"DB_BIBLIOTHEQUE".Mobile[#index].Pos[0].Entr1_Ap_Pos[0] := "I_RPF_TRBV01";
	"DB_BIBLIOTHEQUE".Mobile[#index].Pos[0].Sort0[0] := "I_CO_TRBV01";
	"DB_BIBLIOTHEQUE".Mobile[#index].Pos[0].Sort0_Pr_Fin_Pos[0] := "I_CO_TRBV01";

	//position ouverture
	"DB_BIBLIOTHEQUE".Mobile[#index].Pos[1].Entr0_Ap_Pos[0] := "I_RPF_TRBV01";
	"DB_BIBLIOTHEQUE".Mobile[#index].Pos[1].Entr1_Ap_Pos[0] := "I_RPO_TRBV01";
	"DB_BIBLIOTHEQUE".Mobile[#index].Pos[1].Sort1[0] := "I_CO_TRBV01";
	"DB_BIBLIOTHEQUE".Mobile[#index].Pos[1].Sort0_Pr_Fin_Pos[0] := "I_CO_TRBV01";
	#index := #index + 1;
	(*
	           ╔═══════════╗
	           ║    BV02   ║
	           ╚═══════════╝
	*)
	//++++++++++++++++++++++111++++++++++++++++++++++++++++++\\
	"DB_BIBLIOTHEQUE".Mobile[#index].Nom := 'BV02';





	#index := #index + 1;
	(*
	           ╔═══════════╗
	           ║   TRBV02  ║
	           ╚═══════════╝
	*)
	//++++++++++++++++++++++112++++++++++++++++++++++++++++++\\

	"DB_BIBLIOTHEQUE".Mobile[#index].Nom := 'TRBV02';
	"DB_BIBLIOTHEQUE".Mobile[#index].Mob_Prec[0] := "Index_Mobile"('BV02');
	"DB_BIBLIOTHEQUE".Mobile[#index].Tjr_Desasservi := TRUE;
	"DB_BIBLIOTHEQUE".Mobile[#index].Asservi := FALSE;
	"DB_BIBLIOTHEQUE".Mobile[#index].Pos[0].Nom := '_CLOSE';
	"DB_BIBLIOTHEQUE".Mobile[#index].Pos[1].Nom := '_OPEN';

	//position fermeture
	"DB_BIBLIOTHEQUE".Mobile[#index].Pos[0].Entr0_Ap_Pos[0] := "I_RPO_TRBV02";
	"DB_BIBLIOTHEQUE".Mobile[#index].Pos[0].Entr1_Ap_Pos[0] := "I_RPF_TRBV02";
	"DB_BIBLIOTHEQUE".Mobile[#index].Pos[0].Sort0[0] := "I_CO_TRBV02";
	"DB_BIBLIOTHEQUE".Mobile[#index].Pos[0].Sort0_Pr_Fin_Pos[0] := "I_CO_TRBV02";

	//position ouverture
	"DB_BIBLIOTHEQUE".Mobile[#index].Pos[1].Entr0_Ap_Pos[0] := "I_RPF_TRBV02";
	"DB_BIBLIOTHEQUE".Mobile[#index].Pos[1].Entr1_Ap_Pos[0] := "I_RPO_TRBV02";
	"DB_BIBLIOTHEQUE".Mobile[#index].Pos[1].Sort1[0] := "I_CO_TRBV02";
	"DB_BIBLIOTHEQUE".Mobile[#index].Pos[1].Sort0_Pr_Fin_Pos[0] := "I_CO_TRBV02";
	#index := #index + 1;
	(*
	           ╔═══════════╗
	           ║    BV03   ║
	           ╚═══════════╝
	*)
	//++++++++++++++++++++++113++++++++++++++++++++++++++++++\\
	"DB_BIBLIOTHEQUE".Mobile[#index].Nom := 'BV03';





	#index := #index + 1;
	(*
	           ╔═══════════╗
	           ║   TRBV03  ║
	           ╚═══════════╝
	*)
	//++++++++++++++++++++++114++++++++++++++++++++++++++++++\\

	"DB_BIBLIOTHEQUE".Mobile[#index].Nom := 'TRBV03';
	"DB_BIBLIOTHEQUE".Mobile[#index].Mob_Prec[0] := "Index_Mobile"('BV03');

	"DB_BIBLIOTHEQUE".Mobile[#index].Pos[0].Nom := '_CLOSE';
	"DB_BIBLIOTHEQUE".Mobile[#index].Pos[1].Nom := '_OPEN';
	"DB_BIBLIOTHEQUE".Mobile[#index].Tjr_Desasservi := TRUE;
	"DB_BIBLIOTHEQUE".Mobile[#index].Asservi := FALSE;


	//position fermeture
	"DB_BIBLIOTHEQUE".Mobile[#index].Pos[0].Entr0_Ap_Pos[0] := "I_RPO_TRBV03";
	"DB_BIBLIOTHEQUE".Mobile[#index].Pos[0].Entr1_Ap_Pos[0] := "I_RPF_TRBV03";
	"DB_BIBLIOTHEQUE".Mobile[#index].Pos[0].Sort0[0] := "I_CO_TRBV03";
	"DB_BIBLIOTHEQUE".Mobile[#index].Pos[0].Sort0_Pr_Fin_Pos[0] := "I_CO_TRBV03";

	//position ouverture
	"DB_BIBLIOTHEQUE".Mobile[#index].Pos[1].Entr0_Ap_Pos[0] := "I_RPF_TRBV03";
	"DB_BIBLIOTHEQUE".Mobile[#index].Pos[1].Entr1_Ap_Pos[0] := "I_RPO_TRBV03";
	"DB_BIBLIOTHEQUE".Mobile[#index].Pos[1].Sort1[0] := "I_CO_TRBV03";
	"DB_BIBLIOTHEQUE".Mobile[#index].Pos[1].Sort0_Pr_Fin_Pos[0] := "I_CO_TRBV03";


	#index := #index + 1;
	(*
	           ╔═══════════╗
	           ║    BV04   ║
	           ╚═══════════╝
	*)
	//++++++++++++++++++++++115++++++++++++++++++++++++++++++\\
	"DB_BIBLIOTHEQUE".Mobile[#index].Nom := 'BV04';





	#index := #index + 1;
	(*
	           ╔═══════════╗
	           ║   TRBV04  ║
	           ╚═══════════╝
	*)
	//++++++++++++++++++++++116++++++++++++++++++++++++++++++\\

	"DB_BIBLIOTHEQUE".Mobile[#index].Nom := 'TRBV04';
	"DB_BIBLIOTHEQUE".Mobile[#index].Mob_Prec[0] := "Index_Mobile"('BV04');

	"DB_BIBLIOTHEQUE".Mobile[#index].Pos[0].Nom := '_CLOSE';
	"DB_BIBLIOTHEQUE".Mobile[#index].Pos[1].Nom := '_OPEN';
	"DB_BIBLIOTHEQUE".Mobile[#index].Tjr_Desasservi := TRUE;
	"DB_BIBLIOTHEQUE".Mobile[#index].Asservi := FALSE;


	//position fermeture
	"DB_BIBLIOTHEQUE".Mobile[#index].Pos[0].Entr0_Ap_Pos[0] := "I_RPO_TRBV04";
	"DB_BIBLIOTHEQUE".Mobile[#index].Pos[0].Entr1_Ap_Pos[0] := "I_RPF_TRBV04";
	"DB_BIBLIOTHEQUE".Mobile[#index].Pos[0].Sort0[0] := "I_CO_TRBV04";
	"DB_BIBLIOTHEQUE".Mobile[#index].Pos[0].Sort0_Pr_Fin_Pos[0] := "I_CO_TRBV04";

	//position ouverture
	"DB_BIBLIOTHEQUE".Mobile[#index].Pos[1].Entr0_Ap_Pos[0] := "I_RPF_TRBV04";
	"DB_BIBLIOTHEQUE".Mobile[#index].Pos[1].Entr1_Ap_Pos[0] := "I_RPO_TRBV04";
	"DB_BIBLIOTHEQUE".Mobile[#index].Pos[1].Sort1[0] := "I_CO_TRBV04";
	"DB_BIBLIOTHEQUE".Mobile[#index].Pos[1].Sort0_Pr_Fin_Pos[0] := "I_CO_TRBV04";


	#index := #index + 1;
	(*
	           ╔═══════════╗
	           ║    BV05   ║
	           ╚═══════════╝
	*)
	//++++++++++++++++++++++117++++++++++++++++++++++++++++++\\
	"DB_BIBLIOTHEQUE".Mobile[#index].Nom := 'BV05';





	#index := #index + 1;
	(*
	           ╔═══════════╗
	           ║   TRBV05  ║
	           ╚═══════════╝
	*)
	//++++++++++++++++++++++118++++++++++++++++++++++++++++++\\

	"DB_BIBLIOTHEQUE".Mobile[#index].Nom := 'TRBV05';
	"DB_BIBLIOTHEQUE".Mobile[#index].Mob_Prec[0] := "Index_Mobile"('BV05');
	"DB_BIBLIOTHEQUE".Mobile[#index].Tjr_Desasservi := TRUE;
	"DB_BIBLIOTHEQUE".Mobile[#index].Asservi := FALSE;
	"DB_BIBLIOTHEQUE".Mobile[#index].Pos[0].Nom := '_CLOSE';
	"DB_BIBLIOTHEQUE".Mobile[#index].Pos[1].Nom := '_OPEN';

	//position fermeture
	"DB_BIBLIOTHEQUE".Mobile[#index].Pos[0].Entr0_Ap_Pos[0] := "I_RPO_TRBV05";
	"DB_BIBLIOTHEQUE".Mobile[#index].Pos[0].Entr1_Ap_Pos[0] := "I_RPF_TRBV05";
	"DB_BIBLIOTHEQUE".Mobile[#index].Pos[0].Sort0[0] := "I_CO_TRBV05";
	"DB_BIBLIOTHEQUE".Mobile[#index].Pos[0].Sort0_Pr_Fin_Pos[0] := "I_CO_TRBV05";

	//position ouverture
	"DB_BIBLIOTHEQUE".Mobile[#index].Pos[1].Entr0_Ap_Pos[0] := "I_RPF_TRBV05";
	"DB_BIBLIOTHEQUE".Mobile[#index].Pos[1].Entr1_Ap_Pos[0] := "I_RPO_TRBV05";
	"DB_BIBLIOTHEQUE".Mobile[#index].Pos[1].Sort1[0] := "I_CO_TRBV05";
	"DB_BIBLIOTHEQUE".Mobile[#index].Pos[1].Sort0_Pr_Fin_Pos[0] := "I_CO_TRBV05";
	#index := #index + 1;
	(*
	           ╔═══════════╗
	           ║    BV06   ║
	           ╚═══════════╝
	*)
	//++++++++++++++++++++++119++++++++++++++++++++++++++++++\\
	"DB_BIBLIOTHEQUE".Mobile[#index].Nom := 'BV06';





	#index := #index + 1;
	(*
	           ╔═══════════╗
	           ║   TRBV06  ║
	           ╚═══════════╝
	*)
	//++++++++++++++++++++++120++++++++++++++++++++++++++++++\\

	"DB_BIBLIOTHEQUE".Mobile[#index].Nom := 'TRBV06';
	"DB_BIBLIOTHEQUE".Mobile[#index].Mob_Prec[0] := "Index_Mobile"('BV06');
	"DB_BIBLIOTHEQUE".Mobile[#index].Tjr_Desasservi := TRUE;
	"DB_BIBLIOTHEQUE".Mobile[#index].Asservi := FALSE;
	"DB_BIBLIOTHEQUE".Mobile[#index].Pos[0].Nom := '_CLOSE';
	"DB_BIBLIOTHEQUE".Mobile[#index].Pos[1].Nom := '_OPEN';

	//position fermeture
	"DB_BIBLIOTHEQUE".Mobile[#index].Pos[0].Entr0_Ap_Pos[0] := "I_RPO_TRBV06";
	"DB_BIBLIOTHEQUE".Mobile[#index].Pos[0].Entr1_Ap_Pos[0] := "I_RPF_TRBV06";
	"DB_BIBLIOTHEQUE".Mobile[#index].Pos[0].Sort0[0] := "I_CO_TRBV06";
	"DB_BIBLIOTHEQUE".Mobile[#index].Pos[0].Sort0_Pr_Fin_Pos[0] := "I_CO_TRBV06";

	//position ouverture
	"DB_BIBLIOTHEQUE".Mobile[#index].Pos[1].Entr0_Ap_Pos[0] := "I_RPF_TRBV06";
	"DB_BIBLIOTHEQUE".Mobile[#index].Pos[1].Entr1_Ap_Pos[0] := "I_RPO_TRBV06";
	"DB_BIBLIOTHEQUE".Mobile[#index].Pos[1].Sort1[0] := "I_CO_TRBV06";
	"DB_BIBLIOTHEQUE".Mobile[#index].Pos[1].Sort0_Pr_Fin_Pos[0] := "I_CO_TRBV06";
	#index := #index + 1;
	(*
	           ╔═══════════╗
	           ║    BV07   ║
	           ╚═══════════╝
	*)
	//++++++++++++++++++++++121++++++++++++++++++++++++++++++\\
	"DB_BIBLIOTHEQUE".Mobile[#index].Nom := 'BV07';





	#index := #index + 1;
	(*
	           ╔═══════════╗
	           ║   TRBV07  ║
	           ╚═══════════╝
	*)
	//++++++++++++++++++++++122++++++++++++++++++++++++++++++\\

	"DB_BIBLIOTHEQUE".Mobile[#index].Nom := 'TRBV07';
	"DB_BIBLIOTHEQUE".Mobile[#index].Mob_Prec[0] := "Index_Mobile"('BV07');

	"DB_BIBLIOTHEQUE".Mobile[#index].Pos[0].Nom := '_CLOSE';
	"DB_BIBLIOTHEQUE".Mobile[#index].Pos[1].Nom := '_OPEN';
	"DB_BIBLIOTHEQUE".Mobile[#index].Tjr_Desasservi := TRUE;
	"DB_BIBLIOTHEQUE".Mobile[#index].Asservi := FALSE;


	//position fermeture
	"DB_BIBLIOTHEQUE".Mobile[#index].Pos[0].Entr0_Ap_Pos[0] := "I_RPO_TRBV07";
	"DB_BIBLIOTHEQUE".Mobile[#index].Pos[0].Entr1_Ap_Pos[0] := "I_RPF_TRBV07";
	"DB_BIBLIOTHEQUE".Mobile[#index].Pos[0].Sort0[0] := "I_CO_TRBV07";
	"DB_BIBLIOTHEQUE".Mobile[#index].Pos[0].Sort0_Pr_Fin_Pos[0] := "I_CO_TRBV07";

	//position ouverture
	"DB_BIBLIOTHEQUE".Mobile[#index].Pos[1].Entr0_Ap_Pos[0] := "I_RPF_TRBV07";
	"DB_BIBLIOTHEQUE".Mobile[#index].Pos[1].Entr1_Ap_Pos[0] := "I_RPO_TRBV07";
	"DB_BIBLIOTHEQUE".Mobile[#index].Pos[1].Sort1[0] := "I_CO_TRBV07";
	"DB_BIBLIOTHEQUE".Mobile[#index].Pos[1].Sort0_Pr_Fin_Pos[0] := "I_CO_TRBV07";


	#index := #index + 1;
	(*
	           ╔═══════════╗
	           ║    BV08   ║
	           ╚═══════════╝
	*)
	//++++++++++++++++++++++123++++++++++++++++++++++++++++++\\
	"DB_BIBLIOTHEQUE".Mobile[#index].Nom := 'BV08';





	#index := #index + 1;
	(*
	           ╔═══════════╗
	           ║   TRBV08  ║
	           ╚═══════════╝
	*)
	//++++++++++++++++++++++124++++++++++++++++++++++++++++++\\

	"DB_BIBLIOTHEQUE".Mobile[#index].Nom := 'TRBV08';
	"DB_BIBLIOTHEQUE".Mobile[#index].Mob_Prec[0] := "Index_Mobile"('BV08');

	"DB_BIBLIOTHEQUE".Mobile[#index].Pos[0].Nom := '_CLOSE';
	"DB_BIBLIOTHEQUE".Mobile[#index].Pos[1].Nom := '_OPEN';
	"DB_BIBLIOTHEQUE".Mobile[#index].Tjr_Desasservi := TRUE;
	"DB_BIBLIOTHEQUE".Mobile[#index].Asservi := FALSE;


	//position fermeture
	"DB_BIBLIOTHEQUE".Mobile[#index].Pos[0].Entr0_Ap_Pos[0] := "I_RPO_TRBV08";
	"DB_BIBLIOTHEQUE".Mobile[#index].Pos[0].Entr1_Ap_Pos[0] := "I_RPF_TRBV08";
	"DB_BIBLIOTHEQUE".Mobile[#index].Pos[0].Sort0[0] := "I_CO_TRBV08";
	"DB_BIBLIOTHEQUE".Mobile[#index].Pos[0].Sort0_Pr_Fin_Pos[0] := "I_CO_TRBV08";

	//position ouverture
	"DB_BIBLIOTHEQUE".Mobile[#index].Pos[1].Entr0_Ap_Pos[0] := "I_RPF_TRBV08";
	"DB_BIBLIOTHEQUE".Mobile[#index].Pos[1].Entr1_Ap_Pos[0] := "I_RPO_TRBV08";
	"DB_BIBLIOTHEQUE".Mobile[#index].Pos[1].Sort1[0] := "I_CO_TRBV08";
	"DB_BIBLIOTHEQUE".Mobile[#index].Pos[1].Sort0_Pr_Fin_Pos[0] := "I_CO_TRBV08";


	#index := #index + 1;
	(*
	           ╔═══════════╗
	           ║    BV09   ║
	           ╚═══════════╝
	*)
	//++++++++++++++++++++++125++++++++++++++++++++++++++++++\\
	"DB_BIBLIOTHEQUE".Mobile[#index].Nom := 'BV09';





	#index := #index + 1;
	(*
	           ╔═══════════╗
	           ║   TRBV09  ║
	           ╚═══════════╝
	*)
	//++++++++++++++++++++++126++++++++++++++++++++++++++++++\\

	"DB_BIBLIOTHEQUE".Mobile[#index].Nom := 'TRBV09';
	"DB_BIBLIOTHEQUE".Mobile[#index].Mob_Prec[0] := "Index_Mobile"('BV09');

	"DB_BIBLIOTHEQUE".Mobile[#index].Pos[0].Nom := '_CLOSE';
	"DB_BIBLIOTHEQUE".Mobile[#index].Pos[1].Nom := '_OPEN';
	"DB_BIBLIOTHEQUE".Mobile[#index].Tjr_Desasservi := TRUE;
	"DB_BIBLIOTHEQUE".Mobile[#index].Asservi := FALSE;


	//position fermeture
	"DB_BIBLIOTHEQUE".Mobile[#index].Pos[0].Entr0_Ap_Pos[0] := "I_RPO_TRBV09";
	"DB_BIBLIOTHEQUE".Mobile[#index].Pos[0].Entr1_Ap_Pos[0] := "I_RPF_TRBV09";
	"DB_BIBLIOTHEQUE".Mobile[#index].Pos[0].Sort0[0] := "I_CO_TRBV09";
	"DB_BIBLIOTHEQUE".Mobile[#index].Pos[0].Sort0_Pr_Fin_Pos[0] := "I_CO_TRBV09";

	//position ouverture
	"DB_BIBLIOTHEQUE".Mobile[#index].Pos[1].Entr0_Ap_Pos[0] := "I_RPF_TRBV09";
	"DB_BIBLIOTHEQUE".Mobile[#index].Pos[1].Entr1_Ap_Pos[0] := "I_RPO_TRBV09";
	"DB_BIBLIOTHEQUE".Mobile[#index].Pos[1].Sort1[0] := "I_CO_TRBV09";
	"DB_BIBLIOTHEQUE".Mobile[#index].Pos[1].Sort0_Pr_Fin_Pos[0] := "I_CO_TRBV09";


	#index := #index + 1;
	(*
	           ╔═══════════╗
	           ║    BV10   ║
	           ╚═══════════╝
	*)
	//++++++++++++++++++++++127++++++++++++++++++++++++++++++\\
	"DB_BIBLIOTHEQUE".Mobile[#index].Nom := 'BV10';





	#index := #index + 1;
	(*
	           ╔═══════════╗
	           ║   TRBV10  ║
	           ╚═══════════╝
	*)
	//++++++++++++++++++++++128++++++++++++++++++++++++++++++\\

	"DB_BIBLIOTHEQUE".Mobile[#index].Nom := 'TRBV10';
	"DB_BIBLIOTHEQUE".Mobile[#index].Mob_Prec[0] := "Index_Mobile"('BV10');
	"DB_BIBLIOTHEQUE".Mobile[#index].Tjr_Desasservi := TRUE;
	"DB_BIBLIOTHEQUE".Mobile[#index].Asservi := FALSE;
	"DB_BIBLIOTHEQUE".Mobile[#index].Pos[0].Nom := '_CLOSE';
	"DB_BIBLIOTHEQUE".Mobile[#index].Pos[1].Nom := '_OPEN';

	//position fermeture
	"DB_BIBLIOTHEQUE".Mobile[#index].Pos[0].Entr0_Ap_Pos[0] := "I_RPO_TRBV10";
	"DB_BIBLIOTHEQUE".Mobile[#index].Pos[0].Entr1_Ap_Pos[0] := "I_RPF_TRBV10";
	"DB_BIBLIOTHEQUE".Mobile[#index].Pos[0].Sort0[0] := "I_CO_TRBV10";
	"DB_BIBLIOTHEQUE".Mobile[#index].Pos[0].Sort0_Pr_Fin_Pos[0] := "I_CO_TRBV10";

	//position ouverture
	"DB_BIBLIOTHEQUE".Mobile[#index].Pos[1].Entr0_Ap_Pos[0] := "I_RPF_TRBV10";
	"DB_BIBLIOTHEQUE".Mobile[#index].Pos[1].Entr1_Ap_Pos[0] := "I_RPO_TRBV10";
	"DB_BIBLIOTHEQUE".Mobile[#index].Pos[1].Sort1[0] := "I_CO_TRBV10";
	"DB_BIBLIOTHEQUE".Mobile[#index].Pos[1].Sort0_Pr_Fin_Pos[0] := "I_CO_TRBV10";

	#index := #index + 1;

	(*
	           ╔═══════════╗
	           ║    BV11   ║
	           ╚═══════════╝
	*)
	//++++++++++++++++++++++129++++++++++++++++++++++++++++++\\
	"DB_BIBLIOTHEQUE".Mobile[#index].Nom := 'BV11';





	#index := #index + 1;
	(*
	           ╔═══════════╗
	           ║   TRBV11  ║
	           ╚═══════════╝
	*)
	//++++++++++++++++++++++130++++++++++++++++++++++++++++++\\

	"DB_BIBLIOTHEQUE".Mobile[#index].Nom := 'TRBV11';
	"DB_BIBLIOTHEQUE".Mobile[#index].Mob_Prec[0] := "Index_Mobile"('BV11');
	"DB_BIBLIOTHEQUE".Mobile[#index].Tjr_Desasservi := TRUE;
	"DB_BIBLIOTHEQUE".Mobile[#index].Asservi := FALSE;
	"DB_BIBLIOTHEQUE".Mobile[#index].Pos[0].Nom := '_CLOSE';
	"DB_BIBLIOTHEQUE".Mobile[#index].Pos[1].Nom := '_OPEN';

	//position fermeture
	"DB_BIBLIOTHEQUE".Mobile[#index].Pos[0].Entr0_Ap_Pos[0] := "I_RPO_TRBV11";
	"DB_BIBLIOTHEQUE".Mobile[#index].Pos[0].Entr1_Ap_Pos[0] := "I_RPF_TRBV11";
	"DB_BIBLIOTHEQUE".Mobile[#index].Pos[0].Sort0[0] := "I_CO_TRBV11";
	"DB_BIBLIOTHEQUE".Mobile[#index].Pos[0].Sort0_Pr_Fin_Pos[0] := "I_CO_TRBV11";

	//position ouverture
	"DB_BIBLIOTHEQUE".Mobile[#index].Pos[1].Entr0_Ap_Pos[0] := "I_RPF_TRBV11";
	"DB_BIBLIOTHEQUE".Mobile[#index].Pos[1].Entr1_Ap_Pos[0] := "I_RPO_TRBV11";
	"DB_BIBLIOTHEQUE".Mobile[#index].Pos[1].Sort1[0] := "I_CO_TRBV11";
	"DB_BIBLIOTHEQUE".Mobile[#index].Pos[1].Sort0_Pr_Fin_Pos[0] := "I_CO_TRBV11";

	#index := #index + 1;
	(*
	           ╔═══════════╗
	           ║    BV12   ║
	           ╚═══════════╝
	*)
	//++++++++++++++++++++++131++++++++++++++++++++++++++++++\\
	"DB_BIBLIOTHEQUE".Mobile[#index].Nom := 'BV12';





	#index := #index + 1;
	(*
	           ╔═══════════╗
	           ║   TRBV12  ║
	           ╚═══════════╝
	*)
	//++++++++++++++++++++++132++++++++++++++++++++++++++++++\\

	"DB_BIBLIOTHEQUE".Mobile[#index].Nom := 'TRBV12';
	"DB_BIBLIOTHEQUE".Mobile[#index].Mob_Prec[0] := "Index_Mobile"('BV12');

	"DB_BIBLIOTHEQUE".Mobile[#index].Pos[0].Nom := '_CLOSE';
	"DB_BIBLIOTHEQUE".Mobile[#index].Pos[1].Nom := '_OPEN';
	"DB_BIBLIOTHEQUE".Mobile[#index].Tjr_Desasservi := TRUE;
	"DB_BIBLIOTHEQUE".Mobile[#index].Asservi := FALSE;


	//position fermeture
	"DB_BIBLIOTHEQUE".Mobile[#index].Pos[0].Entr0_Ap_Pos[0] := "I_RPO_TRBV12";
	"DB_BIBLIOTHEQUE".Mobile[#index].Pos[0].Entr1_Ap_Pos[0] := "I_RPF_TRBV12";
	"DB_BIBLIOTHEQUE".Mobile[#index].Pos[0].Sort0[0] := "I_CO_TRBV12";
	"DB_BIBLIOTHEQUE".Mobile[#index].Pos[0].Sort0_Pr_Fin_Pos[0] := "I_CO_TRBV12";

	//position ouverture
	"DB_BIBLIOTHEQUE".Mobile[#index].Pos[1].Entr0_Ap_Pos[0] := "I_RPF_TRBV12";
	"DB_BIBLIOTHEQUE".Mobile[#index].Pos[1].Entr1_Ap_Pos[0] := "I_RPO_TRBV12";
	"DB_BIBLIOTHEQUE".Mobile[#index].Pos[1].Sort1[0] := "I_CO_TRBV12";
	"DB_BIBLIOTHEQUE".Mobile[#index].Pos[1].Sort0_Pr_Fin_Pos[0] := "I_CO_TRBV12";


	#index := #index + 1;
	(*
	           ╔═══════════╗
	           ║    MG1    ║
	           ╚═══════════╝
	*)
	//++++++++++++++++++++++133++++++++++++++++++++++++++++++\\

	"DB_BIBLIOTHEQUE".Mobile[#index].Nom := 'MG1';
	"DB_BIBLIOTHEQUE".Mobile[#index].Mob_Prec[0] := "Index_Mobile"('TR10');
	"DB_BIBLIOTHEQUE".Mobile[#index].Mob_Suiv[0] := "Index_Mobile"('ER10');
	"DB_BIBLIOTHEQUE".Mobile[#index].Pos[1].Mob_Suiv[0] := "Index_Mobile"('ER10');


	"DB_BIBLIOTHEQUE".Mobile[#index].Pos[0].Nom := '_CLOSE';
	"DB_BIBLIOTHEQUE".Mobile[#index].Pos[1].Nom := '_OPEN';
	#index := #index + 1;
	(*
	           ╔═══════════╗
	           ║    BT01   ║
	           ╚═══════════╝
	*)
	//++++++++++++++++++++++134++++++++++++++++++++++++++++++\\
	"DB_BIBLIOTHEQUE".Mobile[#index].Nom := 'BT01';
	#index := #index + 1;

	(*
	           ╔═══════════╗
	           ║    BT02   ║
	           ╚═══════════╝
	*)
	//++++++++++++++++++++++135++++++++++++++++++++++++++++++\\
	"DB_BIBLIOTHEQUE".Mobile[#index].Nom := 'BT02';
	#index := #index + 1;

	(*
	           ╔═══════════╗
	           ║    BT03   ║
	           ╚═══════════╝
	*)
	//++++++++++++++++++++++136++++++++++++++++++++++++++++++\\
	"DB_BIBLIOTHEQUE".Mobile[#index].Nom := 'BT03';
	#index := #index + 1;

	(*
	           ╔═══════════╗
	           ║    BT04   ║
	           ╚═══════════╝
	*)
	//++++++++++++++++++++++137++++++++++++++++++++++++++++++\\
	"DB_BIBLIOTHEQUE".Mobile[#index].Nom := 'BT04';
	#index := #index + 1;

	(*
	           ╔═══════════╗
	           ║    BT06   ║
	           ╚═══════════╝
	*)
	//++++++++++++++++++++++138++++++++++++++++++++++++++++++\\
	"DB_BIBLIOTHEQUE".Mobile[#index].Nom := 'BT06';
	"DB_BIBLIOTHEQUE".Mobile[#index].Mob_Suiv[0] := "Index_Mobile"('TRPBT06');
	"DB_BIBLIOTHEQUE".Mobile[#index].Pos[0].Nom := 'TRPBT06';
	"DB_BIBLIOTHEQUE".Mobile[#index].Pos[0].Mob_Suiv[0] := "Index_Mobile"('TRPBT06');
	#index := #index + 1;

	(*
	           ╔═══════════╗
	           ║    BT07   ║
	           ╚═══════════╝
	*)
	//++++++++++++++++++++++139++++++++++++++++++++++++++++++\\
	"DB_BIBLIOTHEQUE".Mobile[#index].Nom := 'BT07';
	"DB_BIBLIOTHEQUE".Mobile[#index].Mob_Suiv[0] := "Index_Mobile"('TRPBT07');
	"DB_BIBLIOTHEQUE".Mobile[#index].Pos[0].Nom := 'TRPBT07';
	"DB_BIBLIOTHEQUE".Mobile[#index].Pos[0].Mob_Suiv[0] := "Index_Mobile"('TRPBT07');
	#index := #index + 1;

	(*
	           ╔═══════════╗
	           ║    BT08   ║
	           ╚═══════════╝
	*)
	//++++++++++++++++++++++140++++++++++++++++++++++++++++++\\
	"DB_BIBLIOTHEQUE".Mobile[#index].Nom := 'BT08';
	"DB_BIBLIOTHEQUE".Mobile[#index].Mob_Suiv[0] := "Index_Mobile"('TRPBT08');
	"DB_BIBLIOTHEQUE".Mobile[#index].Pos[0].Nom := 'TRPBT08';
	"DB_BIBLIOTHEQUE".Mobile[#index].Pos[0].Mob_Suiv[0] := "Index_Mobile"('TRPBT08');
	#index := #index + 1;

	(*
	           ╔═══════════╗
	           ║    BT09   ║
	           ╚═══════════╝
	*)
	//++++++++++++++++++++++141++++++++++++++++++++++++++++++\\
	"DB_BIBLIOTHEQUE".Mobile[#index].Nom := 'BT09';
	"DB_BIBLIOTHEQUE".Mobile[#index].Mob_Suiv[0] := "Index_Mobile"('TRPBT09');
	"DB_BIBLIOTHEQUE".Mobile[#index].Pos[0].Nom := 'TRPBT09';
	"DB_BIBLIOTHEQUE".Mobile[#index].Pos[0].Mob_Suiv[0] := "Index_Mobile"('TRPBT09');
	#index := #index + 1;

	(*
	           ╔═══════════╗
	           ║    BT10   ║
	           ╚═══════════╝
	*)
	//++++++++++++++++++++++142++++++++++++++++++++++++++++++\\
	"DB_BIBLIOTHEQUE".Mobile[#index].Nom := 'BT10';
	"DB_BIBLIOTHEQUE".Mobile[#index].Mob_Suiv[0] := "Index_Mobile"('TRPBT10');
	"DB_BIBLIOTHEQUE".Mobile[#index].Pos[0].Nom := 'TRPBT10';
	"DB_BIBLIOTHEQUE".Mobile[#index].Pos[0].Mob_Suiv[0] := "Index_Mobile"('TRPBT10');
	#index := #index + 1;

	(*
	           ╔═══════════╗
	           ║    BT11   ║
	           ╚═══════════╝
	*)
	//++++++++++++++++++++++143++++++++++++++++++++++++++++++\\
	"DB_BIBLIOTHEQUE".Mobile[#index].Nom := 'BT11';
	"DB_BIBLIOTHEQUE".Mobile[#index].Mob_Suiv[0] := "Index_Mobile"('TRPBT11');
	"DB_BIBLIOTHEQUE".Mobile[#index].Pos[0].Nom := 'TRPBT11';
	"DB_BIBLIOTHEQUE".Mobile[#index].Pos[0].Mob_Suiv[0] := "Index_Mobile"('TRPBT11');
	#index := #index + 1;

	(*
	           ╔═══════════╗
	           ║    BT12   ║
	           ╚═══════════╝
	*)
	//++++++++++++++++++++++144++++++++++++++++++++++++++++++\\
	"DB_BIBLIOTHEQUE".Mobile[#index].Nom := 'BT12';
	"DB_BIBLIOTHEQUE".Mobile[#index].Mob_Suiv[0] := "Index_Mobile"('TRPBT12');
	"DB_BIBLIOTHEQUE".Mobile[#index].Pos[0].Nom := 'TRPBT12';
	"DB_BIBLIOTHEQUE".Mobile[#index].Pos[0].Mob_Suiv[0] := "Index_Mobile"('TRPBT12');
	#index := #index + 1;

	(*
	           ╔═══════════╗
	           ║    BT13   ║
	           ╚═══════════╝
	*)
	//++++++++++++++++++++++145++++++++++++++++++++++++++++++\\
	"DB_BIBLIOTHEQUE".Mobile[#index].Nom := 'BT13';
	"DB_BIBLIOTHEQUE".Mobile[#index].Mob_Suiv[0] := "Index_Mobile"('TRPBT13');
	"DB_BIBLIOTHEQUE".Mobile[#index].Pos[0].Nom := 'TRPBT13';
	"DB_BIBLIOTHEQUE".Mobile[#index].Pos[0].Mob_Suiv[0] := "Index_Mobile"('TRPBT13');
	#index := #index + 1;

	(*
	           ╔═══════════╗
	           ║    BT14   ║
	           ╚═══════════╝
	*)
	//++++++++++++++++++++++146++++++++++++++++++++++++++++++\\
	"DB_BIBLIOTHEQUE".Mobile[#index].Nom := 'BT14';
	"DB_BIBLIOTHEQUE".Mobile[#index].Mob_Suiv[0] := "Index_Mobile"('TRPBT14');
	"DB_BIBLIOTHEQUE".Mobile[#index].Pos[0].Nom := 'TRPBT14';
	"DB_BIBLIOTHEQUE".Mobile[#index].Pos[0].Mob_Suiv[0] := "Index_Mobile"('TRPBT14');
	#index := #index + 1;

	(*
	           ╔═══════════╗
	           ║    BT15   ║
	           ╚═══════════╝
	*)
	//++++++++++++++++++++++147++++++++++++++++++++++++++++++\\
	"DB_BIBLIOTHEQUE".Mobile[#index].Nom := 'BT15';
	"DB_BIBLIOTHEQUE".Mobile[#index].Mob_Suiv[0] := "Index_Mobile"('TRPBT15');
	"DB_BIBLIOTHEQUE".Mobile[#index].Pos[0].Nom := 'TRPBT15';
	"DB_BIBLIOTHEQUE".Mobile[#index].Pos[0].Mob_Suiv[0] := "Index_Mobile"('TRPBT15');
	#index := #index + 1;

	(*
	           ╔═══════════╗
	           ║    BT16   ║
	           ╚═══════════╝
	*)
	//++++++++++++++++++++++148++++++++++++++++++++++++++++++\\
	"DB_BIBLIOTHEQUE".Mobile[#index].Nom := 'BT16';
	"DB_BIBLIOTHEQUE".Mobile[#index].Mob_Suiv[0] := "Index_Mobile"('TRPBT16');
	"DB_BIBLIOTHEQUE".Mobile[#index].Pos[0].Nom := 'TRPBT16';
	"DB_BIBLIOTHEQUE".Mobile[#index].Pos[0].Mob_Suiv[0] := "Index_Mobile"('TRPBT16');
	#index := #index + 1;

	(*
	           ╔═══════════╗
	           ║    BT17   ║
	           ╚═══════════╝
	*)
	//++++++++++++++++++++++149++++++++++++++++++++++++++++++\\
	"DB_BIBLIOTHEQUE".Mobile[#index].Nom := 'BT17';
	"DB_BIBLIOTHEQUE".Mobile[#index].Mob_Suiv[0] := "Index_Mobile"('TRPBT17');
	"DB_BIBLIOTHEQUE".Mobile[#index].Pos[0].Nom := 'TRPBT17';
	"DB_BIBLIOTHEQUE".Mobile[#index].Pos[0].Mob_Suiv[0] := "Index_Mobile"('TRPBT17');
	#index := #index + 1;

	(*
	           ╔═══════════╗
	           ║    BT18   ║
	           ╚═══════════╝
	*)
	//++++++++++++++++++++++150++++++++++++++++++++++++++++++\\
	"DB_BIBLIOTHEQUE".Mobile[#index].Nom := 'BT18';
	"DB_BIBLIOTHEQUE".Mobile[#index].Mob_Suiv[0] := "Index_Mobile"('TRPBT18');
	"DB_BIBLIOTHEQUE".Mobile[#index].Pos[0].Nom := 'TRPBT18';
	"DB_BIBLIOTHEQUE".Mobile[#index].Pos[0].Mob_Suiv[0] := "Index_Mobile"('TRPBT18');
	#index := #index + 1;

	(*
	           ╔═══════════╗
	           ║    BT19   ║
	           ╚═══════════╝
	*)
	//++++++++++++++++++++++151++++++++++++++++++++++++++++++\\
	"DB_BIBLIOTHEQUE".Mobile[#index].Nom := 'BT19';
	"DB_BIBLIOTHEQUE".Mobile[#index].Mob_Suiv[0] := "Index_Mobile"('TRPBT19');
	"DB_BIBLIOTHEQUE".Mobile[#index].Pos[0].Nom := 'TRPBT19';
	"DB_BIBLIOTHEQUE".Mobile[#index].Pos[0].Mob_Suiv[0] := "Index_Mobile"('TRPBT19');
	#index := #index + 1;

	(*
	           ╔═══════════╗
	           ║    BT20   ║
	           ╚═══════════╝
	*)
	//++++++++++++++++++++++152++++++++++++++++++++++++++++++\\
	"DB_BIBLIOTHEQUE".Mobile[#index].Nom := 'BT20';
	"DB_BIBLIOTHEQUE".Mobile[#index].Mob_Suiv[0] := "Index_Mobile"('TRPBT20');
	"DB_BIBLIOTHEQUE".Mobile[#index].Pos[0].Nom := 'TRPBT20';
	"DB_BIBLIOTHEQUE".Mobile[#index].Pos[0].Mob_Suiv[0] := "Index_Mobile"('TRPBT20');
	#index := #index + 1;

	(*
	           ╔═══════════╗
	           ║    BT21   ║
	           ╚═══════════╝
	*)
	//++++++++++++++++++++++153++++++++++++++++++++++++++++++\\
	"DB_BIBLIOTHEQUE".Mobile[#index].Nom := 'BT21';
	"DB_BIBLIOTHEQUE".Mobile[#index].Mob_Suiv[0] := "Index_Mobile"('TRPBT21');
	"DB_BIBLIOTHEQUE".Mobile[#index].Pos[0].Nom := 'TRPBT21';
	"DB_BIBLIOTHEQUE".Mobile[#index].Pos[0].Mob_Suiv[0] := "Index_Mobile"('TRPBT21');
	#index := #index + 1;

	(*
	           ╔═══════════╗
	           ║  TRPBT01  ║
	           ╚═══════════╝
	*)
	//++++++++++++++++++++++154++++++++++++++++++++++++++++++\\

	"DB_BIBLIOTHEQUE".Mobile[#index].Nom := 'TRPBT01';
	"DB_BIBLIOTHEQUE".Mobile[#index].Mob_Prec[0] := "Index_Mobile"('BT01');

	"DB_BIBLIOTHEQUE".Mobile[#index].Pos[0].Nom := '_CLOSE';
	"DB_BIBLIOTHEQUE".Mobile[#index].Pos[1].Nom := '_OPEN';
	"DB_BIBLIOTHEQUE".Mobile[#index].Tjr_Desasservi := TRUE;
	"DB_BIBLIOTHEQUE".Mobile[#index].Asservi := FALSE;

	//position fermeture
	"DB_BIBLIOTHEQUE".Mobile[#index].Pos[0].Entr0_Ap_Pos[0] := "I_RPO_TRPBT01";
	"DB_BIBLIOTHEQUE".Mobile[#index].Pos[0].Entr1_Ap_Pos[0] := "I_RPF_TRPBT01";
	"DB_BIBLIOTHEQUE".Mobile[#index].Pos[0].Sort0[0] := "I_CO_TRPBT01";
	"DB_BIBLIOTHEQUE".Mobile[#index].Pos[0].Sort0_Pr_Fin_Pos[0] := "I_CO_TRPBT01";

	//position ouverture
	"DB_BIBLIOTHEQUE".Mobile[#index].Pos[1].Entr0_Ap_Pos[0] := "I_RPF_TRPBT01";
	"DB_BIBLIOTHEQUE".Mobile[#index].Pos[1].Entr1_Ap_Pos[0] := "I_RPO_TRPBT01";
	"DB_BIBLIOTHEQUE".Mobile[#index].Pos[1].Sort1[0] := "I_CO_TRPBT01";
	"DB_BIBLIOTHEQUE".Mobile[#index].Pos[1].Sort0_Pr_Fin_Pos[0] := "I_CO_TRPBT01";

	#index := #index + 1;

	(*
	           ╔═══════════╗
	           ║  TRPBT02  ║
	           ╚═══════════╝
	*)
	//++++++++++++++++++++++155++++++++++++++++++++++++++++++\\

	"DB_BIBLIOTHEQUE".Mobile[#index].Nom := 'TRPBT02';
	"DB_BIBLIOTHEQUE".Mobile[#index].Mob_Prec[0] := "Index_Mobile"('BT02');

	"DB_BIBLIOTHEQUE".Mobile[#index].Pos[0].Nom := '_CLOSE';
	"DB_BIBLIOTHEQUE".Mobile[#index].Pos[1].Nom := '_OPEN';
	"DB_BIBLIOTHEQUE".Mobile[#index].Tjr_Desasservi := TRUE;
	"DB_BIBLIOTHEQUE".Mobile[#index].Asservi := FALSE;

	//position fermeture
	"DB_BIBLIOTHEQUE".Mobile[#index].Pos[0].Entr0_Ap_Pos[0] := "I_RPO_TRPBT02";
	"DB_BIBLIOTHEQUE".Mobile[#index].Pos[0].Entr1_Ap_Pos[0] := "I_RPF_TRPBT02";
	"DB_BIBLIOTHEQUE".Mobile[#index].Pos[0].Sort0[0] := "I_CO_TRPBT02";
	"DB_BIBLIOTHEQUE".Mobile[#index].Pos[0].Sort0_Pr_Fin_Pos[0] := "I_CO_TRPBT02";

	//position ouverture
	"DB_BIBLIOTHEQUE".Mobile[#index].Pos[1].Entr0_Ap_Pos[0] := "I_RPF_TRPBT02";
	"DB_BIBLIOTHEQUE".Mobile[#index].Pos[1].Entr1_Ap_Pos[0] := "I_RPO_TRPBT02";
	"DB_BIBLIOTHEQUE".Mobile[#index].Pos[1].Sort1[0] := "I_CO_TRPBT02";
	"DB_BIBLIOTHEQUE".Mobile[#index].Pos[1].Sort0_Pr_Fin_Pos[0] := "I_CO_TRPBT02";

	#index := #index + 1;


	(*
	           ╔═══════════╗
	           ║  TRPBT03  ║
	           ╚═══════════╝
	*)
	//++++++++++++++++++++++156++++++++++++++++++++++++++++++\\

	"DB_BIBLIOTHEQUE".Mobile[#index].Nom := 'TRPBT03';
	"DB_BIBLIOTHEQUE".Mobile[#index].Mob_Prec[0] := "Index_Mobile"('BT03');

	"DB_BIBLIOTHEQUE".Mobile[#index].Pos[0].Nom := '_CLOSE';
	"DB_BIBLIOTHEQUE".Mobile[#index].Pos[1].Nom := '_OPEN';
	"DB_BIBLIOTHEQUE".Mobile[#index].Tjr_Desasservi := TRUE;
	"DB_BIBLIOTHEQUE".Mobile[#index].Asservi := FALSE;

	//position fermeture
	"DB_BIBLIOTHEQUE".Mobile[#index].Pos[0].Entr0_Ap_Pos[0] := "I_RPO_TRPBT03";
	"DB_BIBLIOTHEQUE".Mobile[#index].Pos[0].Entr1_Ap_Pos[0] := "I_RPF_TRPBT03";
	"DB_BIBLIOTHEQUE".Mobile[#index].Pos[0].Sort0[0] := "I_CO_TRPBT03";
	"DB_BIBLIOTHEQUE".Mobile[#index].Pos[0].Sort0_Pr_Fin_Pos[0] := "I_CO_TRPBT03";

	//position ouverture
	"DB_BIBLIOTHEQUE".Mobile[#index].Pos[1].Entr0_Ap_Pos[0] := "I_RPF_TRPBT03";
	"DB_BIBLIOTHEQUE".Mobile[#index].Pos[1].Entr1_Ap_Pos[0] := "I_RPO_TRPBT03";
	"DB_BIBLIOTHEQUE".Mobile[#index].Pos[1].Sort1[0] := "I_CO_TRPBT03";
	"DB_BIBLIOTHEQUE".Mobile[#index].Pos[1].Sort0_Pr_Fin_Pos[0] := "I_CO_TRPBT03";

	#index := #index + 1;

	(*
	           ╔═══════════╗
	           ║  TRPBT04  ║
	           ╚═══════════╝
	*)
	//++++++++++++++++++++++157++++++++++++++++++++++++++++++\\

	"DB_BIBLIOTHEQUE".Mobile[#index].Nom := 'TRPBT04';
	"DB_BIBLIOTHEQUE".Mobile[#index].Mob_Prec[0] := "Index_Mobile"('BT04');

	"DB_BIBLIOTHEQUE".Mobile[#index].Pos[0].Nom := '_CLOSE';
	"DB_BIBLIOTHEQUE".Mobile[#index].Pos[1].Nom := '_OPEN';
	"DB_BIBLIOTHEQUE".Mobile[#index].Tjr_Desasservi := TRUE;
	"DB_BIBLIOTHEQUE".Mobile[#index].Asservi := FALSE;

	//position fermeture
	"DB_BIBLIOTHEQUE".Mobile[#index].Pos[0].Entr0_Ap_Pos[0] := "I_RPO_TRPBT04";
	"DB_BIBLIOTHEQUE".Mobile[#index].Pos[0].Entr1_Ap_Pos[0] := "I_RPF_TRPBT04";
	"DB_BIBLIOTHEQUE".Mobile[#index].Pos[0].Sort0[0] := "I_CO_TRPBT04";
	"DB_BIBLIOTHEQUE".Mobile[#index].Pos[0].Sort0_Pr_Fin_Pos[0] := "I_CO_TRPBT04";

	//position ouverture
	"DB_BIBLIOTHEQUE".Mobile[#index].Pos[1].Entr0_Ap_Pos[0] := "I_RPF_TRPBT04";
	"DB_BIBLIOTHEQUE".Mobile[#index].Pos[1].Entr1_Ap_Pos[0] := "I_RPO_TRPBT04";
	"DB_BIBLIOTHEQUE".Mobile[#index].Pos[1].Sort1[0] := "I_CO_TRPBT04";
	"DB_BIBLIOTHEQUE".Mobile[#index].Pos[1].Sort0_Pr_Fin_Pos[0] := "I_CO_TRPBT04";

	#index := #index + 1;

	(*
	           ╔═══════════╗
	           ║  TRPBT06  ║
	           ╚═══════════╝
	*)
	//++++++++++++++++++++++158++++++++++++++++++++++++++++++\\

	"DB_BIBLIOTHEQUE".Mobile[#index].Nom := 'TRPBT06';
	"DB_BIBLIOTHEQUE".Mobile[#index].Mob_Suiv[0] := "Index_Mobile"('T45');
	"DB_BIBLIOTHEQUE".Mobile[#index].Mob_Prec[0] := "Index_Mobile"('BT06');

	"DB_BIBLIOTHEQUE".Mobile[#index].Pos[0].Nom := '_CLOSE';
	//"DB_BIBLIOTHEQUE".Mobile[#index].Pos[0].Mob_Suiv[0] := "Index_Mobile"('');
	"DB_BIBLIOTHEQUE".Mobile[#index].Pos[1].Nom := '_OPEN';
	"DB_BIBLIOTHEQUE".Mobile[#index].Pos[1].Mob_Suiv[0] := "Index_Mobile"('T45');


	//position fermeture
	"DB_BIBLIOTHEQUE".Mobile[#index].Pos[0].Entr0_Ap_Pos[0] := "I_RPO_TRPBT06";
	"DB_BIBLIOTHEQUE".Mobile[#index].Pos[0].Entr1_Ap_Pos[0] := "I_RPF_TRPBT06";
	"DB_BIBLIOTHEQUE".Mobile[#index].Pos[0].Sort0[0] := "I_CO_TRPBT06";
	"DB_BIBLIOTHEQUE".Mobile[#index].Pos[0].Sort0_Pr_Fin_Pos[0] := "I_CO_TRPBT06";

	//position ouverture
	"DB_BIBLIOTHEQUE".Mobile[#index].Pos[1].Entr0_Ap_Pos[0] := "I_RPF_TRPBT06";
	"DB_BIBLIOTHEQUE".Mobile[#index].Pos[1].Entr1_Ap_Pos[0] := "I_RPO_TRPBT06";
	"DB_BIBLIOTHEQUE".Mobile[#index].Pos[1].Sort1[0] := "I_CO_TRPBT06";
	"DB_BIBLIOTHEQUE".Mobile[#index].Pos[1].Sort0_Pr_Fin_Pos[0] := "I_CO_TRPBT06";


	#index := #index + 1;

	(*
	           ╔═══════════╗
	           ║  TRPBT07  ║
	           ╚═══════════╝
	*)
	//++++++++++++++++++++++159++++++++++++++++++++++++++++++\\

	"DB_BIBLIOTHEQUE".Mobile[#index].Nom := 'TRPBT07';
	"DB_BIBLIOTHEQUE".Mobile[#index].Mob_Suiv[0] := "Index_Mobile"('T45');
	"DB_BIBLIOTHEQUE".Mobile[#index].Mob_Prec[0] := "Index_Mobile"('BT07');

	"DB_BIBLIOTHEQUE".Mobile[#index].Pos[0].Nom := '_CLOSE';
	//"DB_BIBLIOTHEQUE".Mobile[#index].Pos[0].Mob_Suiv[0] := "Index_Mobile"('');
	"DB_BIBLIOTHEQUE".Mobile[#index].Pos[1].Nom := '_OPEN';
	"DB_BIBLIOTHEQUE".Mobile[#index].Pos[1].Mob_Suiv[0] := "Index_Mobile"('T45');


	//position fermeture
	"DB_BIBLIOTHEQUE".Mobile[#index].Pos[0].Entr0_Ap_Pos[0] := "I_RPO_TRPBT07";
	"DB_BIBLIOTHEQUE".Mobile[#index].Pos[0].Entr1_Ap_Pos[0] := "I_RPF_TRPBT07";
	"DB_BIBLIOTHEQUE".Mobile[#index].Pos[0].Sort0[0] := "I_CO_TRPBT07";
	"DB_BIBLIOTHEQUE".Mobile[#index].Pos[0].Sort0_Pr_Fin_Pos[0] := "I_CO_TRPBT07";

	//position ouverture
	"DB_BIBLIOTHEQUE".Mobile[#index].Pos[1].Entr0_Ap_Pos[0] := "I_RPF_TRPBT07";
	"DB_BIBLIOTHEQUE".Mobile[#index].Pos[1].Entr1_Ap_Pos[0] := "I_RPO_TRPBT07";
	"DB_BIBLIOTHEQUE".Mobile[#index].Pos[1].Sort1[0] := "I_CO_TRPBT07";
	"DB_BIBLIOTHEQUE".Mobile[#index].Pos[1].Sort0_Pr_Fin_Pos[0] := "I_CO_TRPBT07";


	#index := #index + 1;

	(*
	           ╔═══════════╗
	           ║  TRPBT08  ║
	           ╚═══════════╝
	*)
	//++++++++++++++++++++++160++++++++++++++++++++++++++++++\\

	"DB_BIBLIOTHEQUE".Mobile[#index].Nom := 'TRPBT08';
	"DB_BIBLIOTHEQUE".Mobile[#index].Mob_Suiv[0] := "Index_Mobile"('T45');
	"DB_BIBLIOTHEQUE".Mobile[#index].Mob_Prec[0] := "Index_Mobile"('BT08');

	"DB_BIBLIOTHEQUE".Mobile[#index].Pos[0].Nom := '_CLOSE';
	//"DB_BIBLIOTHEQUE".Mobile[#index].Pos[0].Mob_Suiv[0] := "Index_Mobile"('');
	"DB_BIBLIOTHEQUE".Mobile[#index].Pos[1].Nom := '_OPEN';
	"DB_BIBLIOTHEQUE".Mobile[#index].Pos[1].Mob_Suiv[0] := "Index_Mobile"('T45');


	//position fermeture
	"DB_BIBLIOTHEQUE".Mobile[#index].Pos[0].Entr0_Ap_Pos[0] := "I_RPO_TRPBT08";
	"DB_BIBLIOTHEQUE".Mobile[#index].Pos[0].Entr1_Ap_Pos[0] := "I_RPF_TRPBT08";
	"DB_BIBLIOTHEQUE".Mobile[#index].Pos[0].Sort0[0] := "I_CO_TRPBT08";
	"DB_BIBLIOTHEQUE".Mobile[#index].Pos[0].Sort0_Pr_Fin_Pos[0] := "I_CO_TRPBT08";

	//position ouverture
	"DB_BIBLIOTHEQUE".Mobile[#index].Pos[1].Entr0_Ap_Pos[0] := "I_RPF_TRPBT08";
	"DB_BIBLIOTHEQUE".Mobile[#index].Pos[1].Entr1_Ap_Pos[0] := "I_RPO_TRPBT08";
	"DB_BIBLIOTHEQUE".Mobile[#index].Pos[1].Sort1[0] := "I_CO_TRPBT08";
	"DB_BIBLIOTHEQUE".Mobile[#index].Pos[1].Sort0_Pr_Fin_Pos[0] := "I_CO_TRPBT08";


	#index := #index + 1;

	(*
	           ╔═══════════╗
	           ║  TRPBT09  ║
	           ╚═══════════╝
	*)
	//++++++++++++++++++++++161++++++++++++++++++++++++++++++\\

	"DB_BIBLIOTHEQUE".Mobile[#index].Nom := 'TRPBT09';
	"DB_BIBLIOTHEQUE".Mobile[#index].Mob_Suiv[0] := "Index_Mobile"('T45');
	"DB_BIBLIOTHEQUE".Mobile[#index].Mob_Prec[0] := "Index_Mobile"('BT09');

	"DB_BIBLIOTHEQUE".Mobile[#index].Pos[0].Nom := '_CLOSE';
	//"DB_BIBLIOTHEQUE".Mobile[#index].Pos[0].Mob_Suiv[0] := "Index_Mobile"('');
	"DB_BIBLIOTHEQUE".Mobile[#index].Pos[1].Nom := '_OPEN';
	"DB_BIBLIOTHEQUE".Mobile[#index].Pos[1].Mob_Suiv[0] := "Index_Mobile"('T45');


	//position fermeture
	"DB_BIBLIOTHEQUE".Mobile[#index].Pos[0].Entr0_Ap_Pos[0] := "I_RPO_TRPBT09";
	"DB_BIBLIOTHEQUE".Mobile[#index].Pos[0].Entr1_Ap_Pos[0] := "I_RPF_TRPBT09";
	"DB_BIBLIOTHEQUE".Mobile[#index].Pos[0].Sort0[0] := "I_CO_TRPBT09";
	"DB_BIBLIOTHEQUE".Mobile[#index].Pos[0].Sort0_Pr_Fin_Pos[0] := "I_CO_TRPBT09";

	//position ouverture
	"DB_BIBLIOTHEQUE".Mobile[#index].Pos[1].Entr0_Ap_Pos[0] := "I_RPF_TRPBT09";
	"DB_BIBLIOTHEQUE".Mobile[#index].Pos[1].Entr1_Ap_Pos[0] := "I_RPO_TRPBT09";
	"DB_BIBLIOTHEQUE".Mobile[#index].Pos[1].Sort1[0] := "I_CO_TRPBT09";
	"DB_BIBLIOTHEQUE".Mobile[#index].Pos[1].Sort0_Pr_Fin_Pos[0] := "I_CO_TRPBT09";


	#index := #index + 1;

	(*
	           ╔═══════════╗
	           ║  TRPBT10  ║
	           ╚═══════════╝
	*)
	//++++++++++++++++++++++162++++++++++++++++++++++++++++++\\

	"DB_BIBLIOTHEQUE".Mobile[#index].Nom := 'TRPBT10';
	"DB_BIBLIOTHEQUE".Mobile[#index].Mob_Suiv[0] := "Index_Mobile"('T51');
	"DB_BIBLIOTHEQUE".Mobile[#index].Mob_Prec[0] := "Index_Mobile"('BT10');

	"DB_BIBLIOTHEQUE".Mobile[#index].Pos[0].Nom := '_CLOSE';
	//"DB_BIBLIOTHEQUE".Mobile[#index].Pos[0].Mob_Suiv[0] := "Index_Mobile"('');
	"DB_BIBLIOTHEQUE".Mobile[#index].Pos[1].Nom := '_OPEN';
	"DB_BIBLIOTHEQUE".Mobile[#index].Pos[1].Mob_Suiv[0] := "Index_Mobile"('T51');


	//position fermeture
	"DB_BIBLIOTHEQUE".Mobile[#index].Pos[0].Entr0_Ap_Pos[0] := "I_RPO_TRPBT10";
	"DB_BIBLIOTHEQUE".Mobile[#index].Pos[0].Entr1_Ap_Pos[0] := "I_RPF_TRPBT10";
	"DB_BIBLIOTHEQUE".Mobile[#index].Pos[0].Sort0[0] := "I_CO_TRPBT10";
	"DB_BIBLIOTHEQUE".Mobile[#index].Pos[0].Sort0_Pr_Fin_Pos[0] := "I_CO_TRPBT10";

	//position ouverture
	"DB_BIBLIOTHEQUE".Mobile[#index].Pos[1].Entr0_Ap_Pos[0] := "I_RPF_TRPBT10";
	"DB_BIBLIOTHEQUE".Mobile[#index].Pos[1].Entr1_Ap_Pos[0] := "I_RPO_TRPBT10";
	"DB_BIBLIOTHEQUE".Mobile[#index].Pos[1].Sort1[0] := "I_CO_TRPBT10";
	"DB_BIBLIOTHEQUE".Mobile[#index].Pos[1].Sort0_Pr_Fin_Pos[0] := "I_CO_TRPBT10";


	#index := #index + 1;

	(*
	           ╔═══════════╗
	           ║  TRPBT11  ║
	           ╚═══════════╝
	*)
	//++++++++++++++++++++++163++++++++++++++++++++++++++++++\\

	"DB_BIBLIOTHEQUE".Mobile[#index].Nom := 'TRPBT11';
	"DB_BIBLIOTHEQUE".Mobile[#index].Mob_Suiv[0] := "Index_Mobile"('T47');
	"DB_BIBLIOTHEQUE".Mobile[#index].Mob_Prec[0] := "Index_Mobile"('BT11');

	"DB_BIBLIOTHEQUE".Mobile[#index].Pos[0].Nom := '_CLOSE';
	//"DB_BIBLIOTHEQUE".Mobile[#index].Pos[0].Mob_Suiv[0] := "Index_Mobile"('');
	"DB_BIBLIOTHEQUE".Mobile[#index].Pos[1].Nom := '_OPEN';
	"DB_BIBLIOTHEQUE".Mobile[#index].Pos[1].Mob_Suiv[0] := "Index_Mobile"('T47');


	//position fermeture
	"DB_BIBLIOTHEQUE".Mobile[#index].Pos[0].Entr0_Ap_Pos[0] := "I_RPO_TRPBT11";
	"DB_BIBLIOTHEQUE".Mobile[#index].Pos[0].Entr1_Ap_Pos[0] := "I_RPF_TRPBT11";
	"DB_BIBLIOTHEQUE".Mobile[#index].Pos[0].Sort0[0] := "I_CO_TRPBT11";
	"DB_BIBLIOTHEQUE".Mobile[#index].Pos[0].Sort0_Pr_Fin_Pos[0] := "I_CO_TRPBT11";

	//position ouverture
	"DB_BIBLIOTHEQUE".Mobile[#index].Pos[1].Entr0_Ap_Pos[0] := "I_RPF_TRPBT11";
	"DB_BIBLIOTHEQUE".Mobile[#index].Pos[1].Entr1_Ap_Pos[0] := "I_RPO_TRPBT11";
	"DB_BIBLIOTHEQUE".Mobile[#index].Pos[1].Sort1[0] := "I_CO_TRPBT11";
	"DB_BIBLIOTHEQUE".Mobile[#index].Pos[1].Sort0_Pr_Fin_Pos[0] := "I_CO_TRPBT11";


	#index := #index + 1;

	(*
	           ╔═══════════╗
	           ║  TRPBT12  ║
	           ╚═══════════╝
	*)
	//++++++++++++++++++++++164++++++++++++++++++++++++++++++\\

	"DB_BIBLIOTHEQUE".Mobile[#index].Nom := 'TRPBT12';
	"DB_BIBLIOTHEQUE".Mobile[#index].Mob_Suiv[0] := "Index_Mobile"('T51');
	"DB_BIBLIOTHEQUE".Mobile[#index].Mob_Prec[0] := "Index_Mobile"('BT12');

	"DB_BIBLIOTHEQUE".Mobile[#index].Pos[0].Nom := '_CLOSE';
	//"DB_BIBLIOTHEQUE".Mobile[#index].Pos[0].Mob_Suiv[0] := "Index_Mobile"('');
	"DB_BIBLIOTHEQUE".Mobile[#index].Pos[1].Nom := '_OPEN';
	"DB_BIBLIOTHEQUE".Mobile[#index].Pos[1].Mob_Suiv[0] := "Index_Mobile"('T51');


	//position fermeture
	"DB_BIBLIOTHEQUE".Mobile[#index].Pos[0].Entr0_Ap_Pos[0] := "I_RPO_TRPBT12";
	"DB_BIBLIOTHEQUE".Mobile[#index].Pos[0].Entr1_Ap_Pos[0] := "I_RPF_TRPBT12";
	"DB_BIBLIOTHEQUE".Mobile[#index].Pos[0].Sort0[0] := "I_CO_TRPBT12";
	"DB_BIBLIOTHEQUE".Mobile[#index].Pos[0].Sort0_Pr_Fin_Pos[0] := "I_CO_TRPBT12";

	//position ouverture
	"DB_BIBLIOTHEQUE".Mobile[#index].Pos[1].Entr0_Ap_Pos[0] := "I_RPF_TRPBT12";
	"DB_BIBLIOTHEQUE".Mobile[#index].Pos[1].Entr1_Ap_Pos[0] := "I_RPO_TRPBT12";
	"DB_BIBLIOTHEQUE".Mobile[#index].Pos[1].Sort1[0] := "I_CO_TRPBT12";
	"DB_BIBLIOTHEQUE".Mobile[#index].Pos[1].Sort0_Pr_Fin_Pos[0] := "I_CO_TRPBT12";


	#index := #index + 1;

	(*
	           ╔═══════════╗
	           ║  TRPBT13  ║
	           ╚═══════════╝
	*)
	//++++++++++++++++++++++165++++++++++++++++++++++++++++++\\

	"DB_BIBLIOTHEQUE".Mobile[#index].Nom := 'TRPBT13';
	"DB_BIBLIOTHEQUE".Mobile[#index].Mob_Suiv[0] := "Index_Mobile"('T47');
	"DB_BIBLIOTHEQUE".Mobile[#index].Mob_Prec[0] := "Index_Mobile"('BT13');

	"DB_BIBLIOTHEQUE".Mobile[#index].Pos[0].Nom := '_CLOSE';
	//"DB_BIBLIOTHEQUE".Mobile[#index].Pos[0].Mob_Suiv[0] := "Index_Mobile"('');
	"DB_BIBLIOTHEQUE".Mobile[#index].Pos[1].Nom := '_OPEN';
	"DB_BIBLIOTHEQUE".Mobile[#index].Pos[1].Mob_Suiv[0] := "Index_Mobile"('T47');


	//position fermeture
	"DB_BIBLIOTHEQUE".Mobile[#index].Pos[0].Entr0_Ap_Pos[0] := "I_RPO_TRPBT13";
	"DB_BIBLIOTHEQUE".Mobile[#index].Pos[0].Entr1_Ap_Pos[0] := "I_RPF_TRPBT13";
	"DB_BIBLIOTHEQUE".Mobile[#index].Pos[0].Sort0[0] := "I_CO_TRPBT13";
	"DB_BIBLIOTHEQUE".Mobile[#index].Pos[0].Sort0_Pr_Fin_Pos[0] := "I_CO_TRPBT13";

	//position ouverture
	"DB_BIBLIOTHEQUE".Mobile[#index].Pos[1].Entr0_Ap_Pos[0] := "I_RPF_TRPBT13";
	"DB_BIBLIOTHEQUE".Mobile[#index].Pos[1].Entr1_Ap_Pos[0] := "I_RPO_TRPBT13";
	"DB_BIBLIOTHEQUE".Mobile[#index].Pos[1].Sort1[0] := "I_CO_TRPBT13";
	"DB_BIBLIOTHEQUE".Mobile[#index].Pos[1].Sort0_Pr_Fin_Pos[0] := "I_CO_TRPBT13";


	#index := #index + 1;

	(*
	           ╔═══════════╗
	           ║  TRPBT14  ║
	           ╚═══════════╝
	*)
	//++++++++++++++++++++++166++++++++++++++++++++++++++++++\\

	"DB_BIBLIOTHEQUE".Mobile[#index].Nom := 'TRPBT14';
	"DB_BIBLIOTHEQUE".Mobile[#index].Mob_Suiv[0] := "Index_Mobile"('T50');
	"DB_BIBLIOTHEQUE".Mobile[#index].Mob_Prec[0] := "Index_Mobile"('BT14');

	"DB_BIBLIOTHEQUE".Mobile[#index].Pos[0].Nom := '_CLOSE';
	//"DB_BIBLIOTHEQUE".Mobile[#index].Pos[0].Mob_Suiv[0] := "Index_Mobile"('');
	"DB_BIBLIOTHEQUE".Mobile[#index].Pos[1].Nom := '_OPEN';
	"DB_BIBLIOTHEQUE".Mobile[#index].Pos[1].Mob_Suiv[0] := "Index_Mobile"('T50');


	//position fermeture
	"DB_BIBLIOTHEQUE".Mobile[#index].Pos[0].Entr0_Ap_Pos[0] := "I_RPO_TRPBT14";
	"DB_BIBLIOTHEQUE".Mobile[#index].Pos[0].Entr1_Ap_Pos[0] := "I_RPF_TRPBT14";
	"DB_BIBLIOTHEQUE".Mobile[#index].Pos[0].Sort0[0] := "I_CO_TRPBT14";
	"DB_BIBLIOTHEQUE".Mobile[#index].Pos[0].Sort0_Pr_Fin_Pos[0] := "I_CO_TRPBT14";

	//position ouverture
	"DB_BIBLIOTHEQUE".Mobile[#index].Pos[1].Entr0_Ap_Pos[0] := "I_RPF_TRPBT14";
	"DB_BIBLIOTHEQUE".Mobile[#index].Pos[1].Entr1_Ap_Pos[0] := "I_RPO_TRPBT14";
	"DB_BIBLIOTHEQUE".Mobile[#index].Pos[1].Sort1[0] := "I_CO_TRPBT14";
	"DB_BIBLIOTHEQUE".Mobile[#index].Pos[1].Sort0_Pr_Fin_Pos[0] := "I_CO_TRPBT14";


	#index := #index + 1;

	(*
	           ╔═══════════╗
	           ║  TRPBT15  ║
	           ╚═══════════╝
	*)
	//++++++++++++++++++++++167++++++++++++++++++++++++++++++\\

	"DB_BIBLIOTHEQUE".Mobile[#index].Nom := 'TRPBT15';
	"DB_BIBLIOTHEQUE".Mobile[#index].Mob_Suiv[0] := "Index_Mobile"('T50');
	"DB_BIBLIOTHEQUE".Mobile[#index].Mob_Prec[0] := "Index_Mobile"('BT15');

	"DB_BIBLIOTHEQUE".Mobile[#index].Pos[0].Nom := '_CLOSE';
	//"DB_BIBLIOTHEQUE".Mobile[#index].Pos[0].Mob_Suiv[0] := "Index_Mobile"('');
	"DB_BIBLIOTHEQUE".Mobile[#index].Pos[1].Nom := '_OPEN';
	"DB_BIBLIOTHEQUE".Mobile[#index].Pos[1].Mob_Suiv[0] := "Index_Mobile"('T50');


	//position fermeture
	"DB_BIBLIOTHEQUE".Mobile[#index].Pos[0].Entr0_Ap_Pos[0] := "I_RPO_TRPBT15";
	"DB_BIBLIOTHEQUE".Mobile[#index].Pos[0].Entr1_Ap_Pos[0] := "I_RPF_TRPBT15";
	"DB_BIBLIOTHEQUE".Mobile[#index].Pos[0].Sort0[0] := "I_CO_TRPBT15";
	"DB_BIBLIOTHEQUE".Mobile[#index].Pos[0].Sort0_Pr_Fin_Pos[0] := "I_CO_TRPBT15";

	//position ouverture
	"DB_BIBLIOTHEQUE".Mobile[#index].Pos[1].Entr0_Ap_Pos[0] := "I_RPF_TRPBT15";
	"DB_BIBLIOTHEQUE".Mobile[#index].Pos[1].Entr1_Ap_Pos[0] := "I_RPO_TRPBT15";
	"DB_BIBLIOTHEQUE".Mobile[#index].Pos[1].Sort1[0] := "I_CO_TRPBT15";
	"DB_BIBLIOTHEQUE".Mobile[#index].Pos[1].Sort0_Pr_Fin_Pos[0] := "I_CO_TRPBT15";


	#index := #index + 1;

	(*
	           ╔═══════════╗
	           ║  TRPBT16  ║
	           ╚═══════════╝
	*)
	//++++++++++++++++++++++168++++++++++++++++++++++++++++++\\

	"DB_BIBLIOTHEQUE".Mobile[#index].Nom := 'TRPBT16';
	"DB_BIBLIOTHEQUE".Mobile[#index].Mob_Suiv[0] := "Index_Mobile"('T51');
	"DB_BIBLIOTHEQUE".Mobile[#index].Mob_Prec[0] := "Index_Mobile"('BT16');

	"DB_BIBLIOTHEQUE".Mobile[#index].Pos[0].Nom := '_CLOSE';
	"DB_BIBLIOTHEQUE".Mobile[#index].Pos[1].Nom := '_OPEN';
	"DB_BIBLIOTHEQUE".Mobile[#index].Pos[1].Mob_Suiv[0] := "Index_Mobile"('T51');


	//position fermeture
	"DB_BIBLIOTHEQUE".Mobile[#index].Pos[0].Entr0_Ap_Pos[0] := "I_RPO_TRPBT16";
	"DB_BIBLIOTHEQUE".Mobile[#index].Pos[0].Entr1_Ap_Pos[0] := "I_RPF_TRPBT16";
	"DB_BIBLIOTHEQUE".Mobile[#index].Pos[0].Sort0[0] := "I_CO_TRPBT16";
	"DB_BIBLIOTHEQUE".Mobile[#index].Pos[0].Sort0_Pr_Fin_Pos[0] := "I_CO_TRPBT16";

	//position ouverture
	"DB_BIBLIOTHEQUE".Mobile[#index].Pos[1].Entr0_Ap_Pos[0] := "I_RPF_TRPBT16";
	"DB_BIBLIOTHEQUE".Mobile[#index].Pos[1].Entr1_Ap_Pos[0] := "I_RPO_TRPBT16";
	"DB_BIBLIOTHEQUE".Mobile[#index].Pos[1].Sort1[0] := "I_CO_TRPBT16";
	"DB_BIBLIOTHEQUE".Mobile[#index].Pos[1].Sort0_Pr_Fin_Pos[0] := "I_CO_TRPBT16";


	#index := #index + 1;

	(*
	           ╔═══════════╗
	           ║  TRPBT17  ║
	           ╚═══════════╝
	*)
	//++++++++++++++++++++++169++++++++++++++++++++++++++++++\\

	"DB_BIBLIOTHEQUE".Mobile[#index].Nom := 'TRPBT17';
	"DB_BIBLIOTHEQUE".Mobile[#index].Mob_Suiv[0] := "Index_Mobile"('T51');
	"DB_BIBLIOTHEQUE".Mobile[#index].Mob_Prec[0] := "Index_Mobile"('BT17');

	"DB_BIBLIOTHEQUE".Mobile[#index].Pos[0].Nom := '_CLOSE';
	//"DB_BIBLIOTHEQUE".Mobile[#index].Pos[0].Mob_Suiv[0] := "Index_Mobile"('');
	"DB_BIBLIOTHEQUE".Mobile[#index].Pos[1].Nom := '_OPEN';
	"DB_BIBLIOTHEQUE".Mobile[#index].Pos[1].Mob_Suiv[0] := "Index_Mobile"('T51');


	//position fermeture
	"DB_BIBLIOTHEQUE".Mobile[#index].Pos[0].Entr0_Ap_Pos[0] := "I_RPO_TRPBT17";
	"DB_BIBLIOTHEQUE".Mobile[#index].Pos[0].Entr1_Ap_Pos[0] := "I_RPF_TRPBT17";
	"DB_BIBLIOTHEQUE".Mobile[#index].Pos[0].Sort0[0] := "I_CO_TRPBT17";
	"DB_BIBLIOTHEQUE".Mobile[#index].Pos[0].Sort0_Pr_Fin_Pos[0] := "I_CO_TRPBT17";

	//position ouverture
	"DB_BIBLIOTHEQUE".Mobile[#index].Pos[1].Entr0_Ap_Pos[0] := "I_RPF_TRPBT17";
	"DB_BIBLIOTHEQUE".Mobile[#index].Pos[1].Entr1_Ap_Pos[0] := "I_RPO_TRPBT17";
	"DB_BIBLIOTHEQUE".Mobile[#index].Pos[1].Sort1[0] := "I_CO_TRPBT17";
	"DB_BIBLIOTHEQUE".Mobile[#index].Pos[1].Sort0_Pr_Fin_Pos[0] := "I_CO_TRPBT17";


	#index := #index + 1;

	(*
	           ╔═══════════╗
	           ║  TRPBT18  ║
	           ╚═══════════╝
	*)
	//++++++++++++++++++++++170++++++++++++++++++++++++++++++\\

	"DB_BIBLIOTHEQUE".Mobile[#index].Nom := 'TRPBT18';
	"DB_BIBLIOTHEQUE".Mobile[#index].Mob_Suiv[0] := "Index_Mobile"('T50');
	"DB_BIBLIOTHEQUE".Mobile[#index].Mob_Prec[0] := "Index_Mobile"('BT18');

	"DB_BIBLIOTHEQUE".Mobile[#index].Pos[0].Nom := '_CLOSE';
	//"DB_BIBLIOTHEQUE".Mobile[#index].Pos[0].Mob_Suiv[0] := "Index_Mobile"('');
	"DB_BIBLIOTHEQUE".Mobile[#index].Pos[1].Nom := '_OPEN';
	"DB_BIBLIOTHEQUE".Mobile[#index].Pos[1].Mob_Suiv[0] := "Index_Mobile"('T50');


	//position fermeture
	"DB_BIBLIOTHEQUE".Mobile[#index].Pos[0].Entr0_Ap_Pos[0] := "I_RPO_TRPBT18";
	"DB_BIBLIOTHEQUE".Mobile[#index].Pos[0].Entr1_Ap_Pos[0] := "I_RPF_TRPBT18";
	"DB_BIBLIOTHEQUE".Mobile[#index].Pos[0].Sort0[0] := "I_CO_TRPBT18";
	"DB_BIBLIOTHEQUE".Mobile[#index].Pos[0].Sort0_Pr_Fin_Pos[0] := "I_CO_TRPBT18";

	//position ouverture
	"DB_BIBLIOTHEQUE".Mobile[#index].Pos[1].Entr0_Ap_Pos[0] := "I_RPF_TRPBT18";
	"DB_BIBLIOTHEQUE".Mobile[#index].Pos[1].Entr1_Ap_Pos[0] := "I_RPO_TRPBT18";
	"DB_BIBLIOTHEQUE".Mobile[#index].Pos[1].Sort1[0] := "I_CO_TRPBT18";
	"DB_BIBLIOTHEQUE".Mobile[#index].Pos[1].Sort0_Pr_Fin_Pos[0] := "I_CO_TRPBT18";


	#index := #index + 1;

	(*
	           ╔═══════════╗
	           ║  TRPBT19  ║
	           ╚═══════════╝
	*)
	//++++++++++++++++++++++171++++++++++++++++++++++++++++++\\

	"DB_BIBLIOTHEQUE".Mobile[#index].Nom := 'TRPBT19';
	"DB_BIBLIOTHEQUE".Mobile[#index].Mob_Suiv[0] := "Index_Mobile"('T50');
	"DB_BIBLIOTHEQUE".Mobile[#index].Mob_Prec[0] := "Index_Mobile"('BT19');

	"DB_BIBLIOTHEQUE".Mobile[#index].Pos[0].Nom := '_CLOSE';
	//"DB_BIBLIOTHEQUE".Mobile[#index].Pos[0].Mob_Suiv[0] := "Index_Mobile"('');
	"DB_BIBLIOTHEQUE".Mobile[#index].Pos[1].Nom := '_OPEN';
	"DB_BIBLIOTHEQUE".Mobile[#index].Pos[1].Mob_Suiv[0] := "Index_Mobile"('T50');


	//position fermeture
	"DB_BIBLIOTHEQUE".Mobile[#index].Pos[0].Entr0_Ap_Pos[0] := "I_RPO_TRPBT19";
	"DB_BIBLIOTHEQUE".Mobile[#index].Pos[0].Entr1_Ap_Pos[0] := "I_RPF_TRPBT19";
	"DB_BIBLIOTHEQUE".Mobile[#index].Pos[0].Sort0[0] := "I_CO_TRPBT19";
	"DB_BIBLIOTHEQUE".Mobile[#index].Pos[0].Sort0_Pr_Fin_Pos[0] := "I_CO_TRPBT19";

	//position ouverture
	"DB_BIBLIOTHEQUE".Mobile[#index].Pos[1].Entr0_Ap_Pos[0] := "I_RPF_TRPBT19";
	"DB_BIBLIOTHEQUE".Mobile[#index].Pos[1].Entr1_Ap_Pos[0] := "I_RPO_TRPBT19";
	"DB_BIBLIOTHEQUE".Mobile[#index].Pos[1].Sort1[0] := "I_CO_TRPBT19";
	"DB_BIBLIOTHEQUE".Mobile[#index].Pos[1].Sort0_Pr_Fin_Pos[0] := "I_CO_TRPBT19";


	#index := #index + 1;

	(*
	           ╔═══════════╗
	           ║  TRPBT20  ║
	           ╚═══════════╝
	*)
	//++++++++++++++++++++++172++++++++++++++++++++++++++++++\\

	"DB_BIBLIOTHEQUE".Mobile[#index].Nom := 'TRPBT20';
	"DB_BIBLIOTHEQUE".Mobile[#index].Mob_Suiv[0] := "Index_Mobile"('T47');
	"DB_BIBLIOTHEQUE".Mobile[#index].Mob_Prec[0] := "Index_Mobile"('BT20');

	"DB_BIBLIOTHEQUE".Mobile[#index].Pos[0].Nom := '_CLOSE';
	//"DB_BIBLIOTHEQUE".Mobile[#index].Pos[0].Mob_Suiv[0] := "Index_Mobile"('');
	"DB_BIBLIOTHEQUE".Mobile[#index].Pos[1].Nom := '_OPEN';
	"DB_BIBLIOTHEQUE".Mobile[#index].Pos[1].Mob_Suiv[0] := "Index_Mobile"('T47');


	//position fermeture
	"DB_BIBLIOTHEQUE".Mobile[#index].Pos[0].Entr0_Ap_Pos[0] := "I_RPO_TRPBT20";
	"DB_BIBLIOTHEQUE".Mobile[#index].Pos[0].Entr1_Ap_Pos[0] := "I_RPF_TRPBT20";
	"DB_BIBLIOTHEQUE".Mobile[#index].Pos[0].Sort0[0] := "I_CO_TRPBT20";
	"DB_BIBLIOTHEQUE".Mobile[#index].Pos[0].Sort0_Pr_Fin_Pos[0] := "I_CO_TRPBT20";

	//position ouverture
	"DB_BIBLIOTHEQUE".Mobile[#index].Pos[1].Entr0_Ap_Pos[0] := "I_RPF_TRPBT20";
	"DB_BIBLIOTHEQUE".Mobile[#index].Pos[1].Entr1_Ap_Pos[0] := "I_RPO_TRPBT20";
	"DB_BIBLIOTHEQUE".Mobile[#index].Pos[1].Sort1[0] := "I_CO_TRPBT20";
	"DB_BIBLIOTHEQUE".Mobile[#index].Pos[1].Sort0_Pr_Fin_Pos[0] := "I_CO_TRPBT20";


	#index := #index + 1;

	(*
	           ╔═══════════╗
	           ║  TRPBT21  ║
	           ╚═══════════╝
	*)
	//++++++++++++++++++++++173++++++++++++++++++++++++++++++\\

	"DB_BIBLIOTHEQUE".Mobile[#index].Nom := 'TRPBT21';
	"DB_BIBLIOTHEQUE".Mobile[#index].Mob_Suiv[0] := "Index_Mobile"('T47');
	"DB_BIBLIOTHEQUE".Mobile[#index].Mob_Prec[0] := "Index_Mobile"('BT21');

	"DB_BIBLIOTHEQUE".Mobile[#index].Pos[0].Nom := '_CLOSE';
	//"DB_BIBLIOTHEQUE".Mobile[#index].Pos[0].Mob_Suiv[0] := "Index_Mobile"('');
	"DB_BIBLIOTHEQUE".Mobile[#index].Pos[1].Nom := '_OPEN';
	"DB_BIBLIOTHEQUE".Mobile[#index].Pos[1].Mob_Suiv[0] := "Index_Mobile"('T47');


	//position fermeture
	"DB_BIBLIOTHEQUE".Mobile[#index].Pos[0].Entr0_Ap_Pos[0] := "I_RPO_TRPBT21";
	"DB_BIBLIOTHEQUE".Mobile[#index].Pos[0].Entr1_Ap_Pos[0] := "I_RPF_TRPBT21";
	"DB_BIBLIOTHEQUE".Mobile[#index].Pos[0].Sort0[0] := "I_CO_TRPBT21";
	"DB_BIBLIOTHEQUE".Mobile[#index].Pos[0].Sort0_Pr_Fin_Pos[0] := "I_CO_TRPBT21";

	//position ouverture
	"DB_BIBLIOTHEQUE".Mobile[#index].Pos[1].Entr0_Ap_Pos[0] := "I_RPF_TRPBT21";
	"DB_BIBLIOTHEQUE".Mobile[#index].Pos[1].Entr1_Ap_Pos[0] := "I_RPO_TRPBT21";
	"DB_BIBLIOTHEQUE".Mobile[#index].Pos[1].Sort1[0] := "I_CO_TRPBT21";
	"DB_BIBLIOTHEQUE".Mobile[#index].Pos[1].Sort0_Pr_Fin_Pos[0] := "I_CO_TRPBT21";


	#index := #index + 1;

	(*
	           ╔═══════════╗
	           ║  TRP1T51  ║
	           ╚═══════════╝
	*)
	//++++++++++++++++++++++174++++++++++++++++++++++++++++++\\

	"DB_BIBLIOTHEQUE".Mobile[#index].Nom := 'TRP1T51';
	"DB_BIBLIOTHEQUE".Mobile[#index].Mob_Suiv[0] := "Index_Mobile"('T47');
	"DB_BIBLIOTHEQUE".Mobile[#index].Mob_Prec[0] := "Index_Mobile"('T51');

	"DB_BIBLIOTHEQUE".Mobile[#index].Pos[0].Nom := '_CLOSE';
	"DB_BIBLIOTHEQUE".Mobile[#index].Pos[1].Nom := '_OPEN';
	"DB_BIBLIOTHEQUE".Mobile[#index].Pos[1].Mob_Suiv[0] := "Index_Mobile"('T47');


	//position fermeture
	"DB_BIBLIOTHEQUE".Mobile[#index].Pos[0].Entr0_Ap_Pos[0] := "I_RPO_TRP1T51";
	"DB_BIBLIOTHEQUE".Mobile[#index].Pos[0].Entr1_Ap_Pos[0] := "I_RPF_TRP1T51";
	"DB_BIBLIOTHEQUE".Mobile[#index].Pos[0].Sort0[0] := "I_CO_TRP1T51";
	"DB_BIBLIOTHEQUE".Mobile[#index].Pos[0].Sort0_Pr_Fin_Pos[0] := "I_CO_TRP1T51";

	//position ouverture
	"DB_BIBLIOTHEQUE".Mobile[#index].Pos[1].Entr0_Ap_Pos[0] := "I_RPF_TRP1T51";
	"DB_BIBLIOTHEQUE".Mobile[#index].Pos[1].Entr1_Ap_Pos[0] := "I_RPO_TRP1T51";
	"DB_BIBLIOTHEQUE".Mobile[#index].Pos[1].Sort1[0] := "I_CO_TRP1T51";
	"DB_BIBLIOTHEQUE".Mobile[#index].Pos[1].Sort0_Pr_Fin_Pos[0] := "I_CO_TRP1T51";


	#index := #index + 1;

	(*
	           ╔═══════════╗
	           ║  TRP1T47  ║
	           ╚═══════════╝
	*)
	//++++++++++++++++++++++175++++++++++++++++++++++++++++++\\

	"DB_BIBLIOTHEQUE".Mobile[#index].Nom := 'TRP1T47';
	"DB_BIBLIOTHEQUE".Mobile[#index].Mob_Suiv[0] := "Index_Mobile"('E23');
	"DB_BIBLIOTHEQUE".Mobile[#index].Mob_Prec[0] := "Index_Mobile"('T47');

	"DB_BIBLIOTHEQUE".Mobile[#index].Pos[0].Nom := '_CLOSE';
	//"DB_BIBLIOTHEQUE".Mobile[#index].Pos[0].Mob_Suiv[0] := "Index_Mobile"('');
	"DB_BIBLIOTHEQUE".Mobile[#index].Pos[1].Nom := '_OPEN';
	"DB_BIBLIOTHEQUE".Mobile[#index].Pos[1].Mob_Suiv[0] := "Index_Mobile"('E23');


	//position fermeture
	"DB_BIBLIOTHEQUE".Mobile[#index].Pos[0].Entr0_Ap_Pos[0] := "I_RPO_TRP1T47";
	"DB_BIBLIOTHEQUE".Mobile[#index].Pos[0].Entr1_Ap_Pos[0] := "I_RPF_TRP1T47";
	"DB_BIBLIOTHEQUE".Mobile[#index].Pos[0].Sort0[0] := "I_CO_TRP1T47";
	"DB_BIBLIOTHEQUE".Mobile[#index].Pos[0].Sort0_Pr_Fin_Pos[0] := "I_CO_TRP1T47";

	//position ouverture
	"DB_BIBLIOTHEQUE".Mobile[#index].Pos[1].Entr0_Ap_Pos[0] := "I_RPF_TRP1T47";
	"DB_BIBLIOTHEQUE".Mobile[#index].Pos[1].Entr1_Ap_Pos[0] := "I_RPO_TRP1T47";
	"DB_BIBLIOTHEQUE".Mobile[#index].Pos[1].Sort1[0] := "I_CO_TRP1T47";
	"DB_BIBLIOTHEQUE".Mobile[#index].Pos[1].Sort0_Pr_Fin_Pos[0] := "I_CO_TRP1T47";


	#index := #index + 1;

	(*
	           ╔═══════════╗
	           ║    E23    ║
	           ╚═══════════╝
	*)
	//++++++++++++++++++++++176++++++++++++++++++++++++++++++\\

	"DB_BIBLIOTHEQUE".Mobile[#index].Nom := 'E23';
	"DB_BIBLIOTHEQUE".Mobile[#index].Mob_Suiv[0] := "Index_Mobile"('BDE23');
	"DB_BIBLIOTHEQUE".Mobile[#index].Mob_Prec[0] := "Index_Mobile"('TRP1T47');


	"DB_BIBLIOTHEQUE".Mobile[#index].Pos[0].Nom := '_VERS_BDE23';
	"DB_BIBLIOTHEQUE".Mobile[#index].Pos[0].Mob_Suiv[0] := "Index_Mobile"('BDE23');




	// Entrées avant pos
	"DB_BIBLIOTHEQUE".Mobile[#index].Pos[0].Entr0_Av_Pos[0] := "I_RD_DISJ_E23";
	"DB_BIBLIOTHEQUE".Mobile[#index].Pos[0].Entr0_Av_Pos[1] := "I_RD_DBHG_E23";
	"DB_BIBLIOTHEQUE".Mobile[#index].Pos[0].Entr0_Av_Pos[2] := "I_RD_DBHD_E23";
	"DB_BIBLIOTHEQUE".Mobile[#index].Pos[0].Entr0_Av_Pos[3] := "I_RD_DBBG_E23";
	"DB_BIBLIOTHEQUE".Mobile[#index].Pos[0].Entr0_Av_Pos[4] := "I_RD_DBBD_E23";
	// Entrées apres pos
	"DB_BIBLIOTHEQUE".Mobile[#index].Pos[0].Entr0_Ap_Pos[0] := "I_RD_DISJ_E23";
	"DB_BIBLIOTHEQUE".Mobile[#index].Pos[0].Entr0_Ap_Pos[1] := "I_RD_DBHG_E23";
	"DB_BIBLIOTHEQUE".Mobile[#index].Pos[0].Entr0_Ap_Pos[2] := "I_RD_DBHD_E23";
	"DB_BIBLIOTHEQUE".Mobile[#index].Pos[0].Entr0_Ap_Pos[3] := "I_RD_DBBG_E23";
	"DB_BIBLIOTHEQUE".Mobile[#index].Pos[0].Entr0_Ap_Pos[4] := "I_RD_DBBD_E23";

	//"DB_BIBLIOTHEQUE".Mobile[#index].Pos[0].Entr1_Ap_Pos[0] := "I_RR_E23";
	"DB_BIBLIOTHEQUE".Mobile[#index].Pos[0].Entr1_Ap_Pos[1] := "I_RM_E23";


	// Entrées fin pos
	//"DB_BIBLIOTHEQUE".Mobile[#index].Pos[0].Entr0_Ap_Fin_Pos[0]:="I_RM_E23";

	// Sorties
	"DB_BIBLIOTHEQUE".Mobile[#index].Pos[0].Sort1[0] := "I_CM_E23";
	"DB_BIBLIOTHEQUE".Mobile[#index].Pos[0].Sort0_Pr_Fin_Pos[0] := "I_CM_E23";


	#index := #index + 1;

	(*
	           ╔═══════════╗
	           ║    E25    ║
	           ╚═══════════╝
	*)
	//++++++++++++++++++++++177++++++++++++++++++++++++++++++\\

	"DB_BIBLIOTHEQUE".Mobile[#index].Nom := 'E25';
	"DB_BIBLIOTHEQUE".Mobile[#index].Mob_Suiv[0] := "Index_Mobile"('B1E25');
	"DB_BIBLIOTHEQUE".Mobile[#index].Mob_Prec[0] := "Index_Mobile"('T50');
	"DB_BIBLIOTHEQUE".Mobile[#index].Mob_Prec[1] := "Index_Mobile"('T47');

	"DB_BIBLIOTHEQUE".Mobile[#index].Pos[0].Nom := '_VERS_B1E25';
	"DB_BIBLIOTHEQUE".Mobile[#index].Pos[0].Mob_Suiv[0] := "Index_Mobile"('B1E25');




	// Entrées avant pos
	"DB_BIBLIOTHEQUE".Mobile[#index].Pos[0].Entr0_Av_Pos[0] := "I_RD_DISJ_E25";
	"DB_BIBLIOTHEQUE".Mobile[#index].Pos[0].Entr0_Av_Pos[1] := "I_RD_DBHG_E25";
	"DB_BIBLIOTHEQUE".Mobile[#index].Pos[0].Entr0_Av_Pos[2] := "I_RD_DBHD_E25";
	"DB_BIBLIOTHEQUE".Mobile[#index].Pos[0].Entr0_Av_Pos[3] := "I_RD_DBBG_E25";
	"DB_BIBLIOTHEQUE".Mobile[#index].Pos[0].Entr0_Av_Pos[4] := "I_RD_DBBD_E25";
	// Entrées apres pos
	"DB_BIBLIOTHEQUE".Mobile[#index].Pos[0].Entr0_Ap_Pos[0] := "I_RD_DISJ_E25";
	"DB_BIBLIOTHEQUE".Mobile[#index].Pos[0].Entr0_Ap_Pos[1] := "I_RD_DBHG_E25";
	"DB_BIBLIOTHEQUE".Mobile[#index].Pos[0].Entr0_Ap_Pos[2] := "I_RD_DBHD_E25";
	"DB_BIBLIOTHEQUE".Mobile[#index].Pos[0].Entr0_Ap_Pos[3] := "I_RD_DBBG_E25";
	"DB_BIBLIOTHEQUE".Mobile[#index].Pos[0].Entr0_Ap_Pos[4] := "I_RD_DBBD_E25";

	//"DB_BIBLIOTHEQUE".Mobile[#index].Pos[0].Entr1_Ap_Pos[0] := "I_RR_E25";
	"DB_BIBLIOTHEQUE".Mobile[#index].Pos[0].Entr1_Ap_Pos[1] := "I_RM_E25";


	// Entrées fin pos
	//"DB_BIBLIOTHEQUE".Mobile[#index].Pos[0].Entr0_Ap_Fin_Pos[0]:="I_RM_E25";

	// Sorties
	"DB_BIBLIOTHEQUE".Mobile[#index].Pos[0].Sort1[0] := "I_CM_E25";
	"DB_BIBLIOTHEQUE".Mobile[#index].Pos[0].Sort0_Pr_Fin_Pos[0] := "I_CM_E25";


	#index := #index + 1;

	(*
	           ╔═══════════╗
	           ║   BDE23   ║
	           ╚═══════════╝
	*)
	//++++++++++++++++++++++178++++++++++++++++++++++++++++++\\
	"DB_BIBLIOTHEQUE".Mobile[#index].Noeud := TRUE;


	"DB_BIBLIOTHEQUE".Mobile[#index].Nom := 'BDE23';
	"DB_BIBLIOTHEQUE".Mobile[#index].Mob_Suiv[0] := "Index_Mobile"('TRM_ENS1');
	"DB_BIBLIOTHEQUE".Mobile[#index].Mob_Suiv[1] := "Index_Mobile"('PF');
	"DB_BIBLIOTHEQUE".Mobile[#index].Mob_Prec[0] := "Index_Mobile"('E23');


	"DB_BIBLIOTHEQUE".Mobile[#index].Pos[0].Nom := '_VERS_TRM_ENS1';
	"DB_BIBLIOTHEQUE".Mobile[#index].Pos[0].Mob_Suiv[0] := "Index_Mobile"('TRM_ENS1');
	"DB_BIBLIOTHEQUE".Mobile[#index].Pos[1].Nom := '_VERS_PF';
	"DB_BIBLIOTHEQUE".Mobile[#index].Pos[1].Mob_Suiv[0] := "Index_Mobile"('PF');




	//Entrées
	"DB_BIBLIOTHEQUE".Mobile[#index].Pos[0].Entr0_Ap_Pos[0] := "I_RP_BDE23_T48";
	"DB_BIBLIOTHEQUE".Mobile[#index].Pos[0].Entr1_Ap_Pos[0] := "I_RP_BDE23_ENS1";
	"DB_BIBLIOTHEQUE".Mobile[#index].Pos[0].Sort1[0] := "I_CP_BDE23_ENS1";
	"DB_BIBLIOTHEQUE".Mobile[#index].Pos[0].Sort0[0] := "I_CP_BDE23_T48";
	"DB_BIBLIOTHEQUE".Mobile[#index].Pos[0].Sort0_Pr_Fin_Pos[0] := "I_CP_BDE23_T48";
	"DB_BIBLIOTHEQUE".Mobile[#index].Pos[0].Sort0_Pr_Fin_Pos[1] := "I_CP_BDE23_ENS1";

	"DB_BIBLIOTHEQUE".Mobile[#index].Pos[1].Entr0_Ap_Pos[0] := "I_RP_BDE23_ENS1";
	"DB_BIBLIOTHEQUE".Mobile[#index].Pos[1].Entr1_Ap_Pos[0] := "I_RP_BDE23_T48";

	//Sorties
	"DB_BIBLIOTHEQUE".Mobile[#index].Pos[1].Sort1[0] := "I_CP_BDE23_T48";
	"DB_BIBLIOTHEQUE".Mobile[#index].Pos[1].Sort0[0] := "I_CP_BDE23_ENS1";
	"DB_BIBLIOTHEQUE".Mobile[#index].Pos[1].Sort0_Pr_Fin_Pos[0] := "I_CP_BDE23_T48";
	"DB_BIBLIOTHEQUE".Mobile[#index].Pos[1].Sort0_Pr_Fin_Pos[1] := "I_CP_BDE23_ENS1";


	#index := #index + 1;

	(*
	           ╔═══════════╗
	           ║   B1E25   ║
	           ╚═══════════╝
	*)
	//++++++++++++++++++++++179++++++++++++++++++++++++++++++\\
	"DB_BIBLIOTHEQUE".Mobile[#index].Noeud := TRUE;


	"DB_BIBLIOTHEQUE".Mobile[#index].Nom := 'B1E25';
	"DB_BIBLIOTHEQUE".Mobile[#index].Mob_Suiv[0] := "Index_Mobile"('TRM_ENS2');
	"DB_BIBLIOTHEQUE".Mobile[#index].Mob_Suiv[1] := "Index_Mobile"('T53');
	"DB_BIBLIOTHEQUE".Mobile[#index].Mob_Prec[0] := "Index_Mobile"('E25');


	"DB_BIBLIOTHEQUE".Mobile[#index].Pos[0].Nom := '_VERS_TRM_ENS2';
	"DB_BIBLIOTHEQUE".Mobile[#index].Pos[0].Mob_Suiv[0] := "Index_Mobile"('TRM_ENS2');
	"DB_BIBLIOTHEQUE".Mobile[#index].Pos[1].Nom := '_VERS_T53';
	"DB_BIBLIOTHEQUE".Mobile[#index].Pos[1].Mob_Suiv[0] := "Index_Mobile"('T53');




	//Entrées
	"DB_BIBLIOTHEQUE".Mobile[#index].Pos[0].Entr0_Ap_Pos[0] := "I_RP_B1E25_T53";
	"DB_BIBLIOTHEQUE".Mobile[#index].Pos[0].Entr1_Ap_Pos[0] := "I_RP_B1E25_ENS2";
	"DB_BIBLIOTHEQUE".Mobile[#index].Pos[0].Sort1[0] := "I_CP_B1E25_ENS2";
	"DB_BIBLIOTHEQUE".Mobile[#index].Pos[0].Sort0[0] := "I_CP_B1E25_T53";
	"DB_BIBLIOTHEQUE".Mobile[#index].Pos[0].Sort0_Pr_Fin_Pos[0] := "I_CP_B1E25_T53";
	"DB_BIBLIOTHEQUE".Mobile[#index].Pos[0].Sort0_Pr_Fin_Pos[1] := "I_CP_B1E25_ENS2";

	"DB_BIBLIOTHEQUE".Mobile[#index].Pos[1].Entr0_Ap_Pos[1] := "I_RP_B1E25_ENS2";
	"DB_BIBLIOTHEQUE".Mobile[#index].Pos[1].Entr1_Ap_Pos[1] := "I_RP_B1E25_T53";

	//Sorties
	"DB_BIBLIOTHEQUE".Mobile[#index].Pos[1].Sort1[0] := "I_CP_B1E25_T53";
	"DB_BIBLIOTHEQUE".Mobile[#index].Pos[1].Sort0[0] := "I_CP_B1E25_ENS2";
	"DB_BIBLIOTHEQUE".Mobile[#index].Pos[1].Sort0_Pr_Fin_Pos[0] := "I_CP_B1E25_T53";
	"DB_BIBLIOTHEQUE".Mobile[#index].Pos[1].Sort0_Pr_Fin_Pos[1] := "I_CP_B1E25_ENS2";


	#index := #index + 1;

	(*
	           ╔═══════════╗
	           ║    T45    ║
	           ╚═══════════╝
	*)
	//++++++++++++++++++++++180++++++++++++++++++++++++++++++\\
	"DB_BIBLIOTHEQUE".Mobile[#index].Nom := 'T45';
	"DB_BIBLIOTHEQUE".Mobile[#index].Mob_Suiv[0] := "Index_Mobile"('T46');
	"DB_BIBLIOTHEQUE".Mobile[#index].Mob_Prec[0] := "Index_Mobile"('TRPBT06');
	"DB_BIBLIOTHEQUE".Mobile[#index].Mob_Prec[1] := "Index_Mobile"('TRPBT07');
	"DB_BIBLIOTHEQUE".Mobile[#index].Mob_Prec[2] := "Index_Mobile"('TRPBT08');
	"DB_BIBLIOTHEQUE".Mobile[#index].Mob_Prec[3] := "Index_Mobile"('TRPBT09');

	"DB_BIBLIOTHEQUE".Mobile[#index].Pos[0].Nom := '_VERS_T46';
	"DB_BIBLIOTHEQUE".Mobile[#index].Pos[0].Mob_Suiv[0] := "Index_Mobile"('T46');

	//"DB_BIBLIOTHEQUE".Mobile[#index].Pass_Mat := "RPM_T45";


	// Entrées avant pos
	"DB_BIBLIOTHEQUE".Mobile[#index].Pos[0].Entr0_Av_Pos[0] := "I_RD_DISJ_T45";
	// Entrées apres pos
	//"DB_BIBLIOTHEQUE".Mobile[#index].Pos[0].Entr0_Ap_Pos[0] := "I_RB_T45";
	"DB_BIBLIOTHEQUE".Mobile[#index].Pos[0].Entr0_Ap_Pos[0] := "I_RD_DISJ_T45";

	//"DB_BIBLIOTHEQUE".Mobile[#index].Pos[0].Entr1_Ap_Pos[0] := "I_RR_T45";
	"DB_BIBLIOTHEQUE".Mobile[#index].Pos[0].Entr1_Ap_Pos[0] := "I_RM_T45";

	// Entrées fin pos
	//"DB_BIBLIOTHEQUE".Mobile[#index].Pos[0].Entr0_Ap_Fin_Pos[0]:="I_RM_T45";

	// Sorties
	"DB_BIBLIOTHEQUE".Mobile[#index].Pos[0].Sort1[0] := "I_CM_T45";
	"DB_BIBLIOTHEQUE".Mobile[#index].Pos[0].Sort0_Pr_Fin_Pos[0] := "I_CM_T45";


	#index := #index + 1;

	(*
	           ╔═══════════╗
	           ║    T46    ║
	           ╚═══════════╝
	*)
	//++++++++++++++++++++++181++++++++++++++++++++++++++++++\\

	"DB_BIBLIOTHEQUE".Mobile[#index].Nom := 'T46';
	"DB_BIBLIOTHEQUE".Mobile[#index].Mob_Suiv[0] := "Index_Mobile"('TRM_ENS1');
	"DB_BIBLIOTHEQUE".Mobile[#index].Mob_Prec[0] := "Index_Mobile"('T45');
	"DB_BIBLIOTHEQUE".Mobile[#index].Pos[0].Nom := '_VERS_TRM_ENS1';
	"DB_BIBLIOTHEQUE".Mobile[#index].Pos[0].Mob_Suiv[0] := "Index_Mobile"('TRM_ENS1');

	//"DB_BIBLIOTHEQUE".Mobile[#index].Pass_Mat := "RPM_T46";


	// Entrées avant pos
	"DB_BIBLIOTHEQUE".Mobile[#index].Pos[0].Entr0_Av_Pos[0] := "I_RD_DISJ_T46";
	// Entrées apres pos
	//"DB_BIBLIOTHEQUE".Mobile[#index].Pos[0].Entr0_Ap_Pos[0] := "I_RB_T46";
	"DB_BIBLIOTHEQUE".Mobile[#index].Pos[0].Entr0_Ap_Pos[0] := "I_RD_DISJ_T46";

	//"DB_BIBLIOTHEQUE".Mobile[#index].Pos[0].Entr1_Ap_Pos[0] := "I_RR_T46";
	"DB_BIBLIOTHEQUE".Mobile[#index].Pos[0].Entr1_Ap_Pos[0] := "I_RM_T46";

	// Entrées fin pos
	//"DB_BIBLIOTHEQUE".Mobile[#index].Pos[0].Entr0_Ap_Fin_Pos[0]:="I_RM_T46";

	// Sorties
	"DB_BIBLIOTHEQUE".Mobile[#index].Pos[0].Sort1[0] := "I_CM_T46";
	"DB_BIBLIOTHEQUE".Mobile[#index].Pos[0].Sort0_Pr_Fin_Pos[0] := "I_CM_T46";


	#index := #index + 1;

	(*
	           ╔═══════════╗
	           ║    T47    ║
	           ╚═══════════╝
	*)
	//++++++++++++++++++++++182++++++++++++++++++++++++++++++\\
	"DB_BIBLIOTHEQUE".Mobile[#index].Noeud := TRUE;


	"DB_BIBLIOTHEQUE".Mobile[#index].Nom := 'T47';
	"DB_BIBLIOTHEQUE".Mobile[#index].Mob_Suiv[0] := "Index_Mobile"('E25');
	"DB_BIBLIOTHEQUE".Mobile[#index].Mob_Suiv[1] := "Index_Mobile"('TRP1T47');


	"DB_BIBLIOTHEQUE".Mobile[#index].Mob_Prec[0] := "Index_Mobile"('TRP1T51');
	"DB_BIBLIOTHEQUE".Mobile[#index].Mob_Prec[1] := "Index_Mobile"('TRPBT13');
	"DB_BIBLIOTHEQUE".Mobile[#index].Mob_Prec[2] := "Index_Mobile"('TRPBT11');
	"DB_BIBLIOTHEQUE".Mobile[#index].Mob_Prec[3] := "Index_Mobile"('TRPBT21');
	"DB_BIBLIOTHEQUE".Mobile[#index].Mob_Prec[4] := "Index_Mobile"('TRPBT20');

	"DB_BIBLIOTHEQUE".Mobile[#index].Pos[0].Nom := '_E25_TRP1T47';
	"DB_BIBLIOTHEQUE".Mobile[#index].Pos[0].Mob_Suiv[0] := "Index_Mobile"('E25');
	"DB_BIBLIOTHEQUE".Mobile[#index].Pos[0].Mob_Suiv[1] := "Index_Mobile"('TRP1T47');


	//"DB_BIBLIOTHEQUE".Mobile[#index].Pass_Mat := "RPM_T47";


	// Entrées avant pos
	"DB_BIBLIOTHEQUE".Mobile[#index].Pos[0].Entr0_Av_Pos[0] := "I_RD_DISJ_T47";
	// Entrées apres pos
	//"DB_BIBLIOTHEQUE".Mobile[#index].Pos[0].Entr0_Ap_Pos[0] := "I_RB_T47";
	"DB_BIBLIOTHEQUE".Mobile[#index].Pos[0].Entr0_Ap_Pos[0] := "I_RD_DISJ_T47";

	//"DB_BIBLIOTHEQUE".Mobile[#index].Pos[0].Entr1_Ap_Pos[0] := "I_RR_T47";
	"DB_BIBLIOTHEQUE".Mobile[#index].Pos[0].Entr1_Ap_Pos[1] := "I_RM_T47";

	// Entrées fin pos
	//"DB_BIBLIOTHEQUE".Mobile[#index].Pos[0].Entr0_Ap_Fin_Pos[0]:="I_RM_T47";

	// Sorties
	"DB_BIBLIOTHEQUE".Mobile[#index].Pos[0].Sort1[0] := "I_CM_T47";
	"DB_BIBLIOTHEQUE".Mobile[#index].Pos[0].Sort0_Pr_Fin_Pos[0] := "I_CM_T47";


	#index := #index + 1;

	(*
	           ╔═══════════╗
	           ║    T50    ║
	           ╚═══════════╝
	*)
	//++++++++++++++++++++++183++++++++++++++++++++++++++++++\\
	"DB_BIBLIOTHEQUE".Mobile[#index].Nom := 'T50';
	"DB_BIBLIOTHEQUE".Mobile[#index].Mob_Suiv[0] := "Index_Mobile"('E25');

	"DB_BIBLIOTHEQUE".Mobile[#index].Mob_Prec[0] := "Index_Mobile"('TRPBT15');
	"DB_BIBLIOTHEQUE".Mobile[#index].Mob_Prec[1] := "Index_Mobile"('TRPBT14');
	"DB_BIBLIOTHEQUE".Mobile[#index].Mob_Prec[2] := "Index_Mobile"('TRPBT18');
	"DB_BIBLIOTHEQUE".Mobile[#index].Mob_Prec[3] := "Index_Mobile"('TRPBT19');

	"DB_BIBLIOTHEQUE".Mobile[#index].Pos[0].Nom := '_VERS_E25';
	"DB_BIBLIOTHEQUE".Mobile[#index].Pos[0].Mob_Suiv[0] := "Index_Mobile"('E25');


	//"DB_BIBLIOTHEQUE".Mobile[#index].Pass_Mat := "RPM_T50";


	// Entrées avant pos
	"DB_BIBLIOTHEQUE".Mobile[#index].Pos[0].Entr0_Av_Pos[0] := "I_RD_DISJ_T50";

	// Entrées apres pos
	//"DB_BIBLIOTHEQUE".Mobile[#index].Pos[0].Entr0_Ap_Pos[0] := "I_RB_T50";
	"DB_BIBLIOTHEQUE".Mobile[#index].Pos[0].Entr0_Ap_Pos[0] := "I_RD_DISJ_T50";


	//"DB_BIBLIOTHEQUE".Mobile[#index].Pos[0].Entr1_Ap_Pos[0] := "I_RR_T50";
	"DB_BIBLIOTHEQUE".Mobile[#index].Pos[0].Entr1_Ap_Pos[0] := "I_RM_T50";

	// Entrées fin pos
	//"DB_BIBLIOTHEQUE".Mobile[#index].Pos[0].Entr0_Ap_Fin_Pos[0]:="I_RM_T50";

	// Sorties
	"DB_BIBLIOTHEQUE".Mobile[#index].Pos[0].Sort1[0] := "I_CM_T50";
	"DB_BIBLIOTHEQUE".Mobile[#index].Pos[0].Sort0_Pr_Fin_Pos[0] := "I_CM_T50";


	#index := #index + 1;

	(*
	           ╔═══════════╗
	           ║    T51    ║
	           ╚═══════════╝
	*)
	//++++++++++++++++++++++184++++++++++++++++++++++++++++++\\
	"DB_BIBLIOTHEQUE".Mobile[#index].Nom := 'T51';
	"DB_BIBLIOTHEQUE".Mobile[#index].Mob_Suiv[0] := "Index_Mobile"('TRP1T51');

	"DB_BIBLIOTHEQUE".Mobile[#index].Mob_Prec[0] := "Index_Mobile"('TRPBT10');
	"DB_BIBLIOTHEQUE".Mobile[#index].Mob_Prec[1] := "Index_Mobile"('TRPBT17');
	"DB_BIBLIOTHEQUE".Mobile[#index].Mob_Prec[2] := "Index_Mobile"('TRPBT16');
	"DB_BIBLIOTHEQUE".Mobile[#index].Mob_Prec[3] := "Index_Mobile"('TRPBT12');

	"DB_BIBLIOTHEQUE".Mobile[#index].Pos[0].Nom := '_VERS_TRP1T51';
	"DB_BIBLIOTHEQUE".Mobile[#index].Pos[0].Mob_Suiv[0] := "Index_Mobile"('TRP1T51');


	//"DB_BIBLIOTHEQUE".Mobile[#index].Pass_Mat := "RPM_T51";


	// Entrées avant pos
	"DB_BIBLIOTHEQUE".Mobile[#index].Pos[0].Entr0_Av_Pos[0] := "I_RD_DISJ_T51";

	// Entrées apres pos
	//"DB_BIBLIOTHEQUE".Mobile[#index].Pos[0].Entr0_Ap_Pos[0] := "I_RB_T51";
	"DB_BIBLIOTHEQUE".Mobile[#index].Pos[0].Entr0_Ap_Pos[0] := "I_RD_DISJ_T51";


	//"DB_BIBLIOTHEQUE".Mobile[#index].Pos[0].Entr1_Ap_Pos[0] := "I_RR_T51";
	"DB_BIBLIOTHEQUE".Mobile[#index].Pos[0].Entr1_Ap_Pos[0] := "I_RM_T51";

	// Entrées fin pos
	//"DB_BIBLIOTHEQUE".Mobile[#index].Pos[0].Entr0_Ap_Fin_Pos[0]:="I_RM_T51";

	// Sorties
	"DB_BIBLIOTHEQUE".Mobile[#index].Pos[0].Sort1[0] := "I_CM_T51";
	"DB_BIBLIOTHEQUE".Mobile[#index].Pos[0].Sort0_Pr_Fin_Pos[0] := "I_CM_T51";


	#index := #index + 1;
	(*
	           ╔═══════════╗
	           ║    T53    ║
	           ╚═══════════╝
	*)
	//++++++++++++++++++++++185++++++++++++++++++++++++++++++\\
	"DB_BIBLIOTHEQUE".Mobile[#index].Nom := 'T53';
	"DB_BIBLIOTHEQUE".Mobile[#index].Noeud := TRUE;
	"DB_BIBLIOTHEQUE".Mobile[#index].Tjr_Desasservi := TRUE;
	"DB_BIBLIOTHEQUE".Mobile[#index].Mob_Prec[0] := "Index_Mobile"('B1E25');



	// "DB_BIBLIOTHEQUE".Mobile[#index].Pass_Mat := "RPM_T53";


	// // Entrées avant pos
	"DB_BIBLIOTHEQUE".Mobile[#index].Pos[0].Entr0_Av_Pos[0] := "I_RD_DISJ_T53";

	// // Entrées apres pos
	// "DB_BIBLIOTHEQUE".Mobile[#index].Pos[0].Entr0_Ap_Pos[0] := "I_RB_T53";
	"DB_BIBLIOTHEQUE".Mobile[#index].Pos[0].Entr0_Ap_Pos[0] := "I_RD_DISJ_T53";


	// "DB_BIBLIOTHEQUE".Mobile[#index].Pos[0].Entr1_Ap_Pos[0] := "I_RR_T53";
	"DB_BIBLIOTHEQUE".Mobile[#index].Pos[0].Entr1_Ap_Pos[0] := "I_RM_T53";

	// // Entrées fin pos
	// //"DB_BIBLIOTHEQUE".Mobile[#index].Pos[0].Entr0_Ap_Fin_Pos[0]:="I_RM_T53";

	// // Sorties
	"DB_BIBLIOTHEQUE".Mobile[#index].Pos[0].Sort1[0] := "I_CM_T53";
	"DB_BIBLIOTHEQUE".Mobile[#index].Pos[0].Sort0_Pr_Fin_Pos[0] := "I_CM_T53";


	#index := #index + 1;
	(*
	           ╔═══════════╗
	           ║  TRM_ENS1 ║
	           ╚═══════════╝
	*)
	//++++++++++++++++++++++186++++++++++++++++++++++++++++++\\
	"DB_BIBLIOTHEQUE".Mobile[#index].Nom := 'TRM_ENS1';
	"DB_BIBLIOTHEQUE".Mobile[#index].Noeud := TRUE;
	"DB_BIBLIOTHEQUE".Mobile[#index].Tjr_Desasservi := TRUE;
	"DB_BIBLIOTHEQUE".Mobile[#index].Mob_Prec[0] := "Index_Mobile"('T46');
	"DB_BIBLIOTHEQUE".Mobile[#index].Mob_Prec[1] := "Index_Mobile"('TRPBT01');
	"DB_BIBLIOTHEQUE".Mobile[#index].Mob_Prec[2] := "Index_Mobile"('TRPBT02');
	"DB_BIBLIOTHEQUE".Mobile[#index].Mob_Prec[3] := "Index_Mobile"('TRPBT03');
	"DB_BIBLIOTHEQUE".Mobile[#index].Mob_Prec[4] := "Index_Mobile"('TRPBT04');
	"DB_BIBLIOTHEQUE".Mobile[#index].Mob_Prec[5] := "Index_Mobile"('BDE23');
	#index := #index + 1;

	(*
	           ╔═══════════╗
	           ║  TRM_ENS2 ║
	           ╚═══════════╝
	*)
	//++++++++++++++++++++++187++++++++++++++++++++++++++++++\\
	"DB_BIBLIOTHEQUE".Mobile[#index].Nom := 'TRM_ENS2';
	"DB_BIBLIOTHEQUE".Mobile[#index].Noeud := TRUE;
	"DB_BIBLIOTHEQUE".Mobile[#index].Tjr_Desasservi := TRUE;
	"DB_BIBLIOTHEQUE".Mobile[#index].Mob_Prec[0] := "Index_Mobile"('B1E25');
	#index := #index + 1;










	//++++++++++++++++++++++++++++++++++++++++++++++++++++++++
	//Renseingnement Deport de Bande et intensite
	(* "DB_DeportBande"."THIS"[0]._DBBD := "E1_DBBD";
	"DB_DeportBande"."THIS"[0]._DBBG := "E1_DBBG";
	"DB_DeportBande"."THIS"[0]._DBHD := "E1_DBHD";
	"DB_DeportBande"."THIS"[0]._DBHG := "E1_DBHG"; *)
	// "DB_CntrlInt"."THIS"[0]._Amperage := "E1_I";



	(* "DB_DeportBande"."THIS"[2]._DBBD := "E4_DBBD";
	"DB_DeportBande"."THIS"[2]._DBBG := "E4_DBBG";
	"DB_DeportBande"."THIS"[2]._DBHD := "E4_DBHD";
	"DB_DeportBande"."THIS"[2]._DBHG := "E4_DBHG"; *)
	// "DB_CntrlInt"."THIS"[0]._Amperage := "E4_I";

	(* "DB_DeportBande"."THIS"[3]._DBBD := "E5_DBBD";
	"DB_DeportBande"."THIS"[3]._DBBG := "E5_DBBG";
	"DB_DeportBande"."THIS"[3]._DBHD := "E5_DBHD";
	"DB_DeportBande"."THIS"[3]._DBHG := "E5_DBHG"; *)
	// "DB_CntrlInt"."THIS"[0]._Amperage := "E5_I";







END_FUNCTION

